REGION Network 1: Режим глобальной симуляции
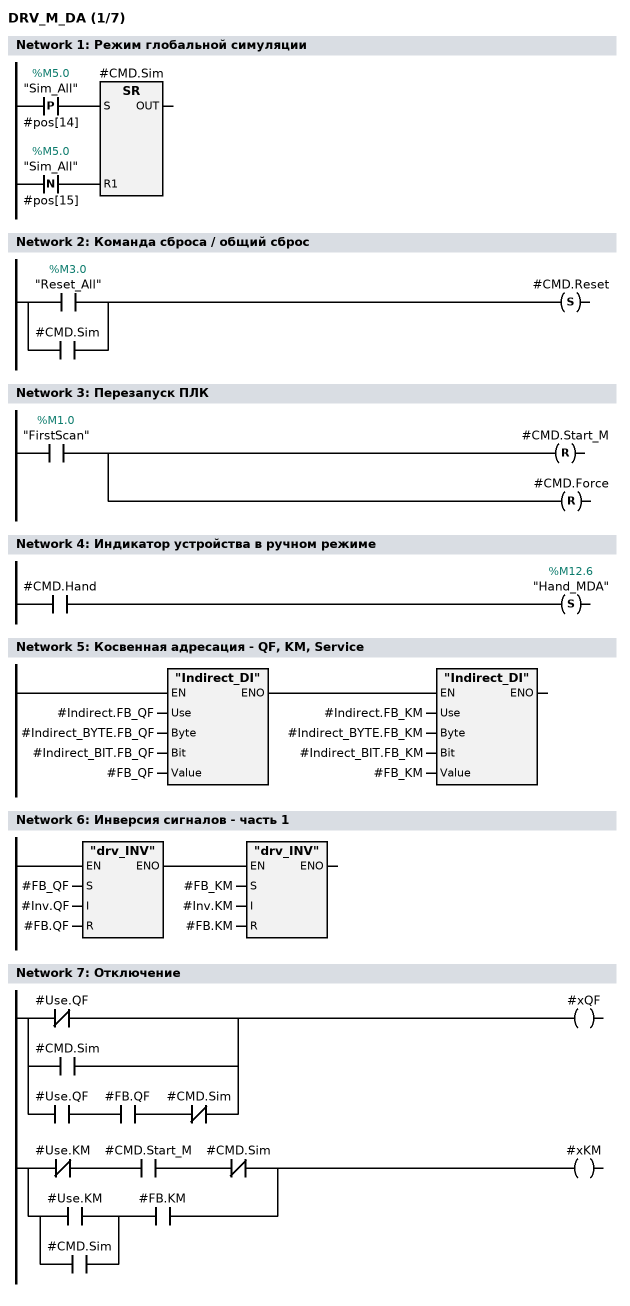
   RUNG wire#powerrail
      P_Contact(operand := "Sim_All", bit := #pos[14])
      S_SR(operand := #CMD.Sim, r1 := wire#w1)
   END_RUNG
   RUNG wire#powerrail
      N_Contact(operand := "Sim_All", bit := #pos[15])
   END_RUNG wire#w1
   // the same network as SCL:
   #_w1 := "Sim_All" AND NOT #pos[14];   // rising edge of "Sim_All"
   #pos[14] := "Sim_All";
   #_w2 := NOT "Sim_All" AND #pos[15];   // falling edge of "Sim_All"
   #pos[15] := "Sim_All";
   IF #_w1 THEN
       #CMD.Sim := TRUE;   // SR flip-flop
   END_IF;
   IF #_w2 THEN #CMD.Sim := FALSE; END_IF;
END_REGION

REGION Network 2: Команда сброса / общий сброс
   RUNG wire#powerrail
      Contact( "Reset_All" )
      wire#w1
      S_Coil( #CMD.Reset )
   END_RUNG
   RUNG wire#powerrail
      Contact( #CMD.Sim )
   END_RUNG wire#w1
   // the same network as SCL:
   IF "Reset_All" OR #CMD.Sim THEN #CMD.Reset := TRUE; END_IF;
END_REGION

REGION Network 3: Перезапуск ПЛК
   RUNG wire#powerrail
      Contact( "FirstScan" )
      wire#w1
      R_Coil( #CMD.Start_M )
   END_RUNG
   RUNG wire#w1
      R_Coil( #CMD.Force )
   END_RUNG
   // the same network as SCL:
   IF "FirstScan" THEN
       #CMD.Start_M := FALSE;
       #CMD.Force := FALSE;
   END_IF;
END_REGION

REGION Network 4: Индикатор устройства в ручном режиме
   RUNG wire#powerrail
      Contact( #CMD.Hand )
      S_Coil( "Hand_MDA" )
   END_RUNG
   // the same network as SCL:
   IF #CMD.Hand THEN "Hand_MDA" := TRUE; END_IF;
END_REGION

REGION Network 5: Косвенная адресация - QF, KM, Service
   RUNG wire#powerrail
      "Indirect_DI"(Use := #Indirect.FB_QF, "Byte" := #Indirect_BYTE.FB_QF, Bit := #Indirect_BIT.FB_QF, Value := #FB_QF)
      "Indirect_DI"(Use := #Indirect.FB_KM, "Byte" := #Indirect_BYTE.FB_KM, Bit := #Indirect_BIT.FB_KM, Value := #FB_KM)
   END_RUNG
   // the same network as SCL:
   "Indirect_DI"(Use := #Indirect.FB_QF,
                 "Byte" := #Indirect_BYTE.FB_QF,
                 Bit := #Indirect_BIT.FB_QF,
                 Value := #FB_QF,
                 ENO => #_w1);
   IF #_w1 THEN
       "Indirect_DI"(Use := #Indirect.FB_KM,
                     "Byte" := #Indirect_BYTE.FB_KM,
                     Bit := #Indirect_BIT.FB_KM,
                     Value := #FB_KM);
   END_IF;
END_REGION

REGION Network 6: Инверсия сигналов - часть 1
   RUNG wire#powerrail
      "drv_INV"(S := #FB_QF, I := #Inv.QF, R := #FB.QF)
      "drv_INV"(S := #FB_KM, I := #Inv.KM, R := #FB.KM)
   END_RUNG
   // the same network as SCL:
   "drv_INV"(S := #FB_QF, I := #Inv.QF, R := #FB.QF, ENO => #_w1);
   IF #_w1 THEN "drv_INV"(S := #FB_KM, I := #Inv.KM, R := #FB.KM); END_IF;
END_REGION

REGION Network 7: Отключение
   RUNG wire#powerrail
      I_Contact( #Use.QF )
      wire#w1
      Coil( #xQF )
   END_RUNG
   RUNG wire#powerrail
      Contact( #CMD.Sim )
   END_RUNG wire#w1
   RUNG wire#powerrail
      Contact( #Use.QF )
      Contact( #FB.QF )
      I_Contact( #CMD.Sim )
   END_RUNG wire#w1
   RUNG wire#powerrail
      I_Contact( #Use.KM )
      Contact( #CMD.Start_M )
      I_Contact( #CMD.Sim )
      wire#w2
      Coil( #xKM )
   END_RUNG
   RUNG wire#powerrail
      Contact( #Use.KM )
      wire#w3
      Contact( #FB.KM )
   END_RUNG wire#w2
   RUNG wire#powerrail
      Contact( #CMD.Sim )
   END_RUNG wire#w3
   // the same network as SCL:
   #xQF := NOT #Use.QF OR #CMD.Sim OR (#Use.QF AND #FB.QF AND NOT #CMD.Sim);
   #xKM := (NOT #Use.KM AND #CMD.Start_M AND NOT #CMD.Sim) OR ((#Use.KM OR #CMD.Sim) AND #FB.KM);
END_REGION

REGION Network 8: Режим работы устройства / определение режима работы
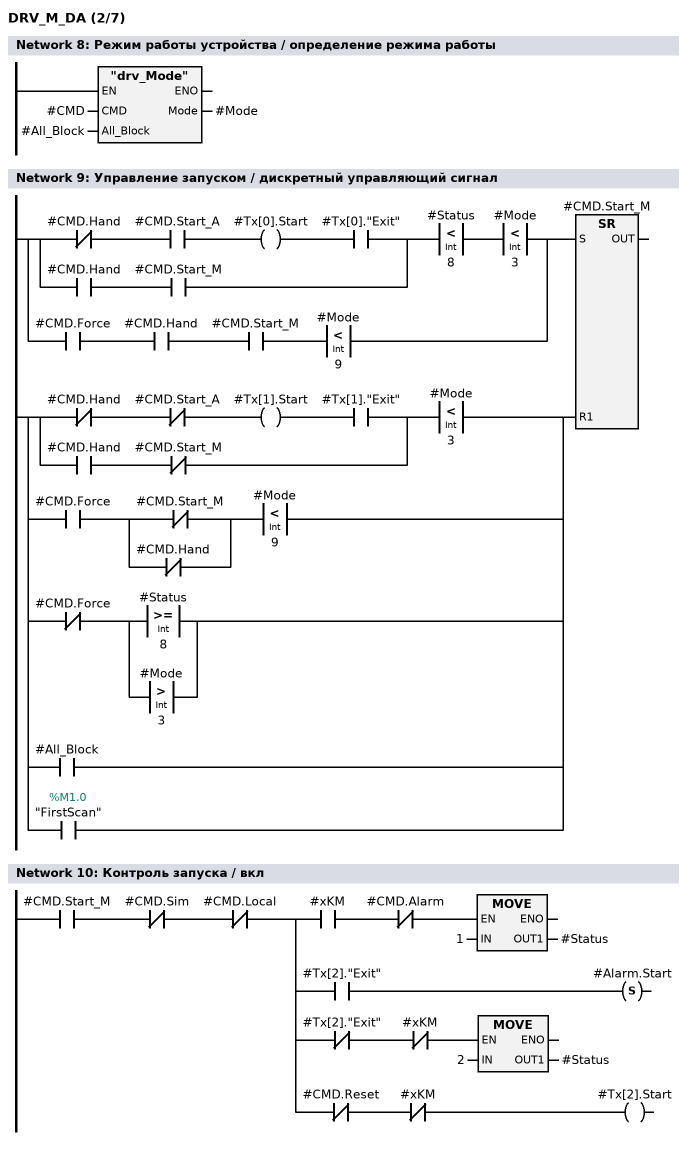
   RUNG wire#powerrail
      "drv_Mode"(CMD := #CMD, All_Block := #All_Block, Mode => #Mode)
   END_RUNG
   // the same network as SCL:
   "drv_Mode"(CMD := #CMD, All_Block := #All_Block, Mode => #Mode);
END_REGION

REGION Network 9: Управление запуском / дискретный управляющий сигнал
   RUNG wire#powerrail
      I_Contact( #CMD.Hand )
      Contact( #CMD.Start_A )
      Coil( #Tx[0].Start )
      Contact( #Tx[0]."Exit" )
      wire#w1
      { S7_Templates := "SrcType := Int" } LT_Contact(in1 := #Status, in2 := 8)
      { S7_Templates := "SrcType := Int" } LT_Contact(in1 := #Mode, in2 := 3)
      wire#w2
      S_SR(operand := #CMD.Start_M, r1 := wire#w7)
   END_RUNG
   RUNG wire#powerrail
      Contact( #CMD.Hand )
      Contact( #CMD.Start_M )
   END_RUNG wire#w1
   RUNG wire#powerrail
      Contact( #CMD.Force )
      Contact( #CMD.Hand )
      Contact( #CMD.Start_M )
      { S7_Templates := "SrcType := Int" } LT_Contact(in1 := #Mode, in2 := 9)
   END_RUNG wire#w2
   RUNG wire#powerrail
      I_Contact( #CMD.Hand )
      I_Contact( #CMD.Start_A )
      Coil( #Tx[1].Start )
      Contact( #Tx[1]."Exit" )
      wire#w3
      { S7_Templates := "SrcType := Int" } LT_Contact(in1 := #Mode, in2 := 3)
   END_RUNG wire#w7
   RUNG wire#powerrail
      Contact( #CMD.Hand )
      I_Contact( #CMD.Start_M )
   END_RUNG wire#w3
   RUNG wire#powerrail
      Contact( #CMD.Force )
      wire#w4
      I_Contact( #CMD.Start_M )
      wire#w5
      { S7_Templates := "SrcType := Int" } LT_Contact(in1 := #Mode, in2 := 9)
   END_RUNG wire#w7
   RUNG wire#w4
      I_Contact( #CMD.Hand )
   END_RUNG wire#w5
   RUNG wire#powerrail
      I_Contact( #CMD.Force )
      wire#w6
      { S7_Templates := "SrcType := Int" } GE_Contact(in1 := #Status, in2 := 8)
   END_RUNG wire#w7
   RUNG wire#w6
      { S7_Templates := "SrcType := Int" } GT_Contact(in1 := #Mode, in2 := 3)
   END_RUNG wire#w7
   RUNG wire#powerrail
      Contact( #All_Block )
   END_RUNG wire#w7
   RUNG wire#powerrail
      Contact( "FirstScan" )
   END_RUNG wire#w7
   // the same network as SCL:
   #Tx[0].Start := NOT #CMD.Hand AND #CMD.Start_A;
   #_w1 := (((NOT #CMD.Hand AND #CMD.Start_A AND #Tx[0]."Exit") OR (#CMD.Hand AND #CMD.Start_M)) AND (#Status < 8) AND (#Mode < 3)) OR (#CMD.Force AND #CMD.Hand AND #CMD.Start_M AND (#Mode < 9));
   #Tx[1].Start := NOT #CMD.Hand AND NOT #CMD.Start_A;
   #_w2 := (((NOT #CMD.Hand AND NOT #CMD.Start_A AND #Tx[1]."Exit") OR (#CMD.Hand AND NOT #CMD.Start_M)) AND (#Mode < 3)) OR (#CMD.Force AND (NOT #CMD.Start_M OR NOT #CMD.Hand) AND (#Mode < 9)) OR (NOT #CMD.Force AND ((#Status >= 8) OR (#Mode > 3))) OR #All_Block OR "FirstScan";
   IF #_w1 THEN
       #CMD.Start_M := TRUE;   // SR flip-flop
   END_IF;
   IF #_w2 THEN #CMD.Start_M := FALSE; END_IF;
END_REGION

REGION Network 10: Контроль запуска / вкл
   RUNG wire#powerrail
      Contact( #CMD.Start_M )
      I_Contact( #CMD.Sim )
      I_Contact( #CMD.Local )
      wire#w1
      Contact( #xKM )
      I_Contact( #CMD.Alarm )
      { S7_GenerateENO := "TRUE" } Move(in := 1, out1 => #Status)
   END_RUNG
   RUNG wire#w1
      Contact( #Tx[2]."Exit" )
      S_Coil( #Alarm.Start )
   END_RUNG
   RUNG wire#w1
      I_Contact( #Tx[2]."Exit" )
      I_Contact( #xKM )
      { S7_GenerateENO := "TRUE" } Move(in := 2, out1 => #Status)
   END_RUNG
   RUNG wire#w1
      I_Contact( #CMD.Reset )
      I_Contact( #xKM )
      Coil( #Tx[2].Start )
   END_RUNG
   // the same network as SCL:
   #_w1 := #CMD.Start_M AND NOT #CMD.Sim AND NOT #CMD.Local;
   IF #_w1 AND #xKM AND NOT #CMD.Alarm THEN #Status := 1; END_IF;
   IF #_w1 AND #Tx[2]."Exit" THEN #Alarm.Start := TRUE; END_IF;
   IF #_w1 AND NOT #Tx[2]."Exit" AND NOT #xKM THEN #Status := 2; END_IF;
   #Tx[2].Start := #_w1 AND NOT #CMD.Reset AND NOT #xKM;
END_REGION

REGION Network 11: Контроль останова / выкл
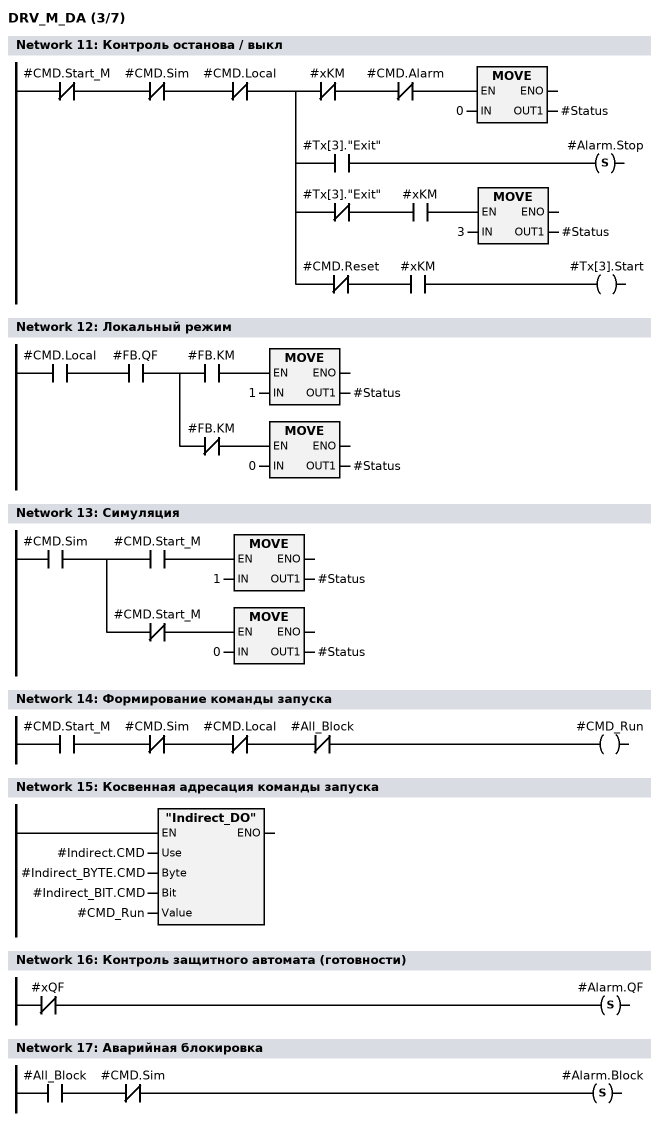
   RUNG wire#powerrail
      I_Contact( #CMD.Start_M )
      I_Contact( #CMD.Sim )
      I_Contact( #CMD.Local )
      wire#w1
      I_Contact( #xKM )
      I_Contact( #CMD.Alarm )
      { S7_GenerateENO := "TRUE" } Move(in := 0, out1 => #Status)
   END_RUNG
   RUNG wire#w1
      Contact( #Tx[3]."Exit" )
      S_Coil( #Alarm.Stop )
   END_RUNG
   RUNG wire#w1
      I_Contact( #Tx[3]."Exit" )
      Contact( #xKM )
      { S7_GenerateENO := "TRUE" } Move(in := 3, out1 => #Status)
   END_RUNG
   RUNG wire#w1
      I_Contact( #CMD.Reset )
      Contact( #xKM )
      Coil( #Tx[3].Start )
   END_RUNG
   // the same network as SCL:
   #_w1 := NOT #CMD.Start_M AND NOT #CMD.Sim AND NOT #CMD.Local;
   IF #_w1 AND NOT #xKM AND NOT #CMD.Alarm THEN #Status := 0; END_IF;
   IF #_w1 AND #Tx[3]."Exit" THEN #Alarm.Stop := TRUE; END_IF;
   IF #_w1 AND NOT #Tx[3]."Exit" AND #xKM THEN #Status := 3; END_IF;
   #Tx[3].Start := #_w1 AND NOT #CMD.Reset AND #xKM;
END_REGION

REGION Network 12: Локальный режим
   RUNG wire#powerrail
      Contact( #CMD.Local )
      Contact( #FB.QF )
      wire#w1
      Contact( #FB.KM )
      { S7_GenerateENO := "TRUE" } Move(in := 1, out1 => #Status)
   END_RUNG
   RUNG wire#w1
      I_Contact( #FB.KM )
      { S7_GenerateENO := "TRUE" } Move(in := 0, out1 => #Status)
   END_RUNG
   // the same network as SCL:
   #_w1 := #CMD.Local AND #FB.QF;
   IF #_w1 AND #FB.KM THEN #Status := 1; END_IF;
   IF #_w1 AND NOT #FB.KM THEN #Status := 0; END_IF;
END_REGION

REGION Network 13: Симуляция
   RUNG wire#powerrail
      Contact( #CMD.Sim )
      wire#w1
      Contact( #CMD.Start_M )
      { S7_GenerateENO := "TRUE" } Move(in := 1, out1 => #Status)
   END_RUNG
   RUNG wire#w1
      I_Contact( #CMD.Start_M )
      { S7_GenerateENO := "TRUE" } Move(in := 0, out1 => #Status)
   END_RUNG
   // the same network as SCL:
   IF #CMD.Sim AND #CMD.Start_M THEN #Status := 1; END_IF;
   IF #CMD.Sim AND NOT #CMD.Start_M THEN #Status := 0; END_IF;
END_REGION

REGION Network 14: Формирование команды запуска
   RUNG wire#powerrail
      Contact( #CMD.Start_M )
      I_Contact( #CMD.Sim )
      I_Contact( #CMD.Local )
      I_Contact( #All_Block )
      Coil( #CMD_Run )
   END_RUNG
   // the same network as SCL:
   #CMD_Run := #CMD.Start_M AND NOT #CMD.Sim AND NOT #CMD.Local AND NOT #All_Block;
END_REGION

REGION Network 15: Косвенная адресация команды запуска
   RUNG wire#powerrail
      "Indirect_DO"(Use := #Indirect.CMD, "Byte" := #Indirect_BYTE.CMD, Bit := #Indirect_BIT.CMD, Value := #CMD_Run)
   END_RUNG
   // the same network as SCL:
   "Indirect_DO"(Use := #Indirect.CMD,
                 "Byte" := #Indirect_BYTE.CMD,
                 Bit := #Indirect_BIT.CMD,
                 Value := #CMD_Run);
END_REGION

REGION Network 16: Контроль защитного автомата (готовности)
   RUNG wire#powerrail
      I_Contact( #xQF )
      S_Coil( #Alarm.QF )
   END_RUNG
   // the same network as SCL:
   IF NOT #xQF THEN #Alarm.QF := TRUE; END_IF;
END_REGION

REGION Network 17: Аварийная блокировка
   RUNG wire#powerrail
      Contact( #All_Block )
      I_Contact( #CMD.Sim )
      S_Coil( #Alarm.Block )
   END_RUNG
   // the same network as SCL:
   IF #All_Block AND NOT #CMD.Sim THEN #Alarm.Block := TRUE; END_IF;
END_REGION

REGION Network 18: Сигнал аварии
   // Safety - сработал датчик безопасности, подключается через отдельный дискретный вход
   // Termo - сработала термозащита, подключается через отдельный дискретный вход
   // Alarm - сработала внешняя авария, подключается через отдельный дискретный вход
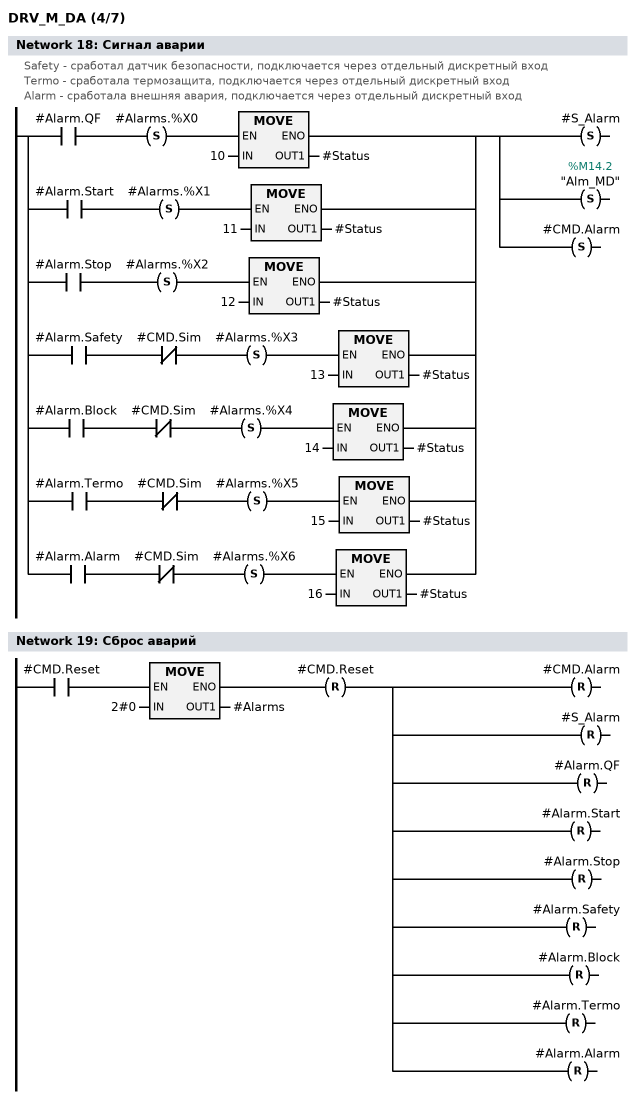
   RUNG wire#powerrail
      Contact( #Alarm.QF )
      S_Coil( #Alarms.%X0 )
      { S7_GenerateENO := "TRUE" } Move(in := 10, out1 => #Status)
      wire#w1
      S_Coil( #S_Alarm )
   END_RUNG
   RUNG wire#powerrail
      Contact( #Alarm.Start )
      S_Coil( #Alarms.%X1 )
      { S7_GenerateENO := "TRUE" } Move(in := 11, out1 => #Status)
   END_RUNG wire#w1
   RUNG wire#powerrail
      Contact( #Alarm.Stop )
      S_Coil( #Alarms.%X2 )
      { S7_GenerateENO := "TRUE" } Move(in := 12, out1 => #Status)
   END_RUNG wire#w1
   RUNG wire#powerrail
      Contact( #Alarm.Safety )
      I_Contact( #CMD.Sim )
      S_Coil( #Alarms.%X3 )
      { S7_GenerateENO := "TRUE" } Move(in := 13, out1 => #Status)
   END_RUNG wire#w1
   RUNG wire#powerrail
      Contact( #Alarm.Block )
      I_Contact( #CMD.Sim )
      S_Coil( #Alarms.%X4 )
      { S7_GenerateENO := "TRUE" } Move(in := 14, out1 => #Status)
   END_RUNG wire#w1
   RUNG wire#powerrail
      Contact( #Alarm.Termo )
      I_Contact( #CMD.Sim )
      S_Coil( #Alarms.%X5 )
      { S7_GenerateENO := "TRUE" } Move(in := 15, out1 => #Status)
   END_RUNG wire#w1
   RUNG wire#powerrail
      Contact( #Alarm.Alarm )
      I_Contact( #CMD.Sim )
      S_Coil( #Alarms.%X6 )
      { S7_GenerateENO := "TRUE" } Move(in := 16, out1 => #Status)
   END_RUNG wire#w1
   RUNG wire#w1
      S_Coil( "Alm_MD" )
   END_RUNG
   RUNG wire#w1
      S_Coil( #CMD.Alarm )
   END_RUNG
   // the same network as SCL:
   // ENO of a box is taken as its EN; it also drops when the box reports an error
   IF #Alarm.QF THEN
       #Alarms.%X0 := TRUE;
       #Status := 10;
   END_IF;
   IF #Alarm.Start THEN
       #Alarms.%X1 := TRUE;
       #Status := 11;
   END_IF;
   IF #Alarm.Stop THEN
       #Alarms.%X2 := TRUE;
       #Status := 12;
   END_IF;
   #_w1 := #Alarm.Safety AND NOT #CMD.Sim;
   IF #_w1 THEN
       #Alarms.%X3 := TRUE;
       #Status := 13;
   END_IF;
   #_w2 := #Alarm.Block AND NOT #CMD.Sim;
   IF #_w2 THEN
       #Alarms.%X4 := TRUE;
       #Status := 14;
   END_IF;
   #_w3 := #Alarm.Termo AND NOT #CMD.Sim;
   IF #_w3 THEN
       #Alarms.%X5 := TRUE;
       #Status := 15;
   END_IF;
   #_w4 := #Alarm.Alarm AND NOT #CMD.Sim;
   IF #_w4 THEN
       #Alarms.%X6 := TRUE;
       #Status := 16;
   END_IF;
   IF #Alarm.QF OR #Alarm.Start OR #Alarm.Stop OR #_w1 OR #_w2 OR #_w3 OR #_w4 THEN
       #S_Alarm := TRUE;
       "Alm_MD" := TRUE;
       #CMD.Alarm := TRUE;
   END_IF;
END_REGION

REGION Network 19: Сброс аварий
   RUNG wire#powerrail
      Contact( #CMD.Reset )
      Move(in := 2#0, out1 => #Alarms)
      R_Coil( #CMD.Reset )
      wire#w1
      R_Coil( #CMD.Alarm )
   END_RUNG
   RUNG wire#w1
      R_Coil( #S_Alarm )
   END_RUNG
   RUNG wire#w1
      R_Coil( #Alarm.QF )
   END_RUNG
   RUNG wire#w1
      R_Coil( #Alarm.Start )
   END_RUNG
   RUNG wire#w1
      R_Coil( #Alarm.Stop )
   END_RUNG
   RUNG wire#w1
      R_Coil( #Alarm.Safety )
   END_RUNG
   RUNG wire#w1
      R_Coil( #Alarm.Block )
   END_RUNG
   RUNG wire#w1
      R_Coil( #Alarm.Termo )
   END_RUNG
   RUNG wire#w1
      R_Coil( #Alarm.Alarm )
   END_RUNG
   // the same network as SCL:
   IF #CMD.Reset THEN #Alarms := 2#0; END_IF;
   #_w1 := #CMD.Reset;
   IF #_w1 THEN
       #CMD.Reset := FALSE;
       #CMD.Alarm := FALSE;
       #S_Alarm := FALSE;
       #Alarm.QF := FALSE;
       #Alarm.Start := FALSE;
       #Alarm.Stop := FALSE;
       #Alarm.Safety := FALSE;
       #Alarm.Block := FALSE;
       #Alarm.Termo := FALSE;
       #Alarm.Alarm := FALSE;
   END_IF;
END_REGION

REGION Network 20: События привода
   // 0 - ручной режим активирован
   // 1 - ручной режим деактивирован
   // 2 - принудительный режим активирован
   // 3 - принудительный режим деактивирован
   // 4 - запуск в ручном режиме
   // 5 - останов в ручном режиме
   // 6 - местный режим управления активирован
   // 7 - местный режим управления деактивирован
   // 8 - запущено в местном режиме
   // 9 - остановлено в местном режиме
   // 10 - сервисный режим активирован
   // 11 - сервисный режим деактивирован
   // 12 - проведено сервисное обслуживание
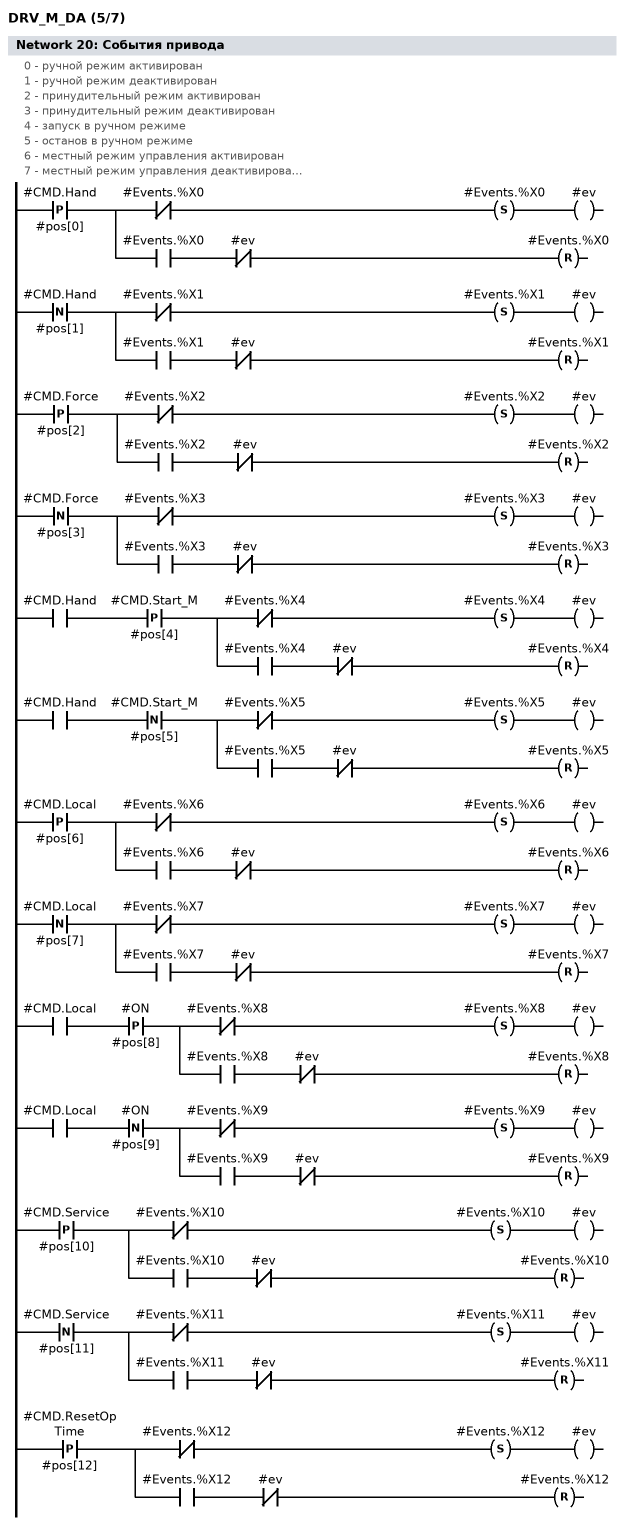
   RUNG wire#powerrail
      P_Contact(operand := #CMD.Hand, bit := #pos[0])
      wire#w1
      I_Contact( #Events.%X0 )
      S_Coil( #Events.%X0 )
      Coil( #ev )
   END_RUNG
   RUNG wire#w1
      Contact( #Events.%X0 )
      I_Contact( #ev )
      R_Coil( #Events.%X0 )
   END_RUNG
   RUNG wire#powerrail
      N_Contact(operand := #CMD.Hand, bit := #pos[1])
      wire#w2
      I_Contact( #Events.%X1 )
      S_Coil( #Events.%X1 )
      Coil( #ev )
   END_RUNG
   RUNG wire#w2
      Contact( #Events.%X1 )
      I_Contact( #ev )
      R_Coil( #Events.%X1 )
   END_RUNG
   RUNG wire#powerrail
      P_Contact(operand := #CMD.Force, bit := #pos[2])
      wire#w3
      I_Contact( #Events.%X2 )
      S_Coil( #Events.%X2 )
      Coil( #ev )
   END_RUNG
   RUNG wire#w3
      Contact( #Events.%X2 )
      I_Contact( #ev )
      R_Coil( #Events.%X2 )
   END_RUNG
   RUNG wire#powerrail
      N_Contact(operand := #CMD.Force, bit := #pos[3])
      wire#w4
      I_Contact( #Events.%X3 )
      S_Coil( #Events.%X3 )
      Coil( #ev )
   END_RUNG
   RUNG wire#w4
      Contact( #Events.%X3 )
      I_Contact( #ev )
      R_Coil( #Events.%X3 )
   END_RUNG
   RUNG wire#powerrail
      Contact( #CMD.Hand )
      P_Contact(operand := #CMD.Start_M, bit := #pos[4])
      wire#w5
      I_Contact( #Events.%X4 )
      S_Coil( #Events.%X4 )
      Coil( #ev )
   END_RUNG
   RUNG wire#w5
      Contact( #Events.%X4 )
      I_Contact( #ev )
      R_Coil( #Events.%X4 )
   END_RUNG
   RUNG wire#powerrail
      Contact( #CMD.Hand )
      N_Contact(operand := #CMD.Start_M, bit := #pos[5])
      wire#w6
      I_Contact( #Events.%X5 )
      S_Coil( #Events.%X5 )
      Coil( #ev )
   END_RUNG
   RUNG wire#w6
      Contact( #Events.%X5 )
      I_Contact( #ev )
      R_Coil( #Events.%X5 )
   END_RUNG
   RUNG wire#powerrail
      P_Contact(operand := #CMD.Local, bit := #pos[6])
      wire#w7
      I_Contact( #Events.%X6 )
      S_Coil( #Events.%X6 )
      Coil( #ev )
   END_RUNG
   RUNG wire#w7
      Contact( #Events.%X6 )
      I_Contact( #ev )
      R_Coil( #Events.%X6 )
   END_RUNG
   RUNG wire#powerrail
      N_Contact(operand := #CMD.Local, bit := #pos[7])
      wire#w8
      I_Contact( #Events.%X7 )
      S_Coil( #Events.%X7 )
      Coil( #ev )
   END_RUNG
   RUNG wire#w8
      Contact( #Events.%X7 )
      I_Contact( #ev )
      R_Coil( #Events.%X7 )
   END_RUNG
   RUNG wire#powerrail
      Contact( #CMD.Local )
      P_Contact(operand := #ON, bit := #pos[8])
      wire#w9
      I_Contact( #Events.%X8 )
      S_Coil( #Events.%X8 )
      Coil( #ev )
   END_RUNG
   RUNG wire#w9
      Contact( #Events.%X8 )
      I_Contact( #ev )
      R_Coil( #Events.%X8 )
   END_RUNG
   RUNG wire#powerrail
      Contact( #CMD.Local )
      N_Contact(operand := #ON, bit := #pos[9])
      wire#w10
      I_Contact( #Events.%X9 )
      S_Coil( #Events.%X9 )
      Coil( #ev )
   END_RUNG
   RUNG wire#w10
      Contact( #Events.%X9 )
      I_Contact( #ev )
      R_Coil( #Events.%X9 )
   END_RUNG
   RUNG wire#powerrail
      P_Contact(operand := #CMD.Service, bit := #pos[10])
      wire#w11
      I_Contact( #Events.%X10 )
      S_Coil( #Events.%X10 )
      Coil( #ev )
   END_RUNG
   RUNG wire#w11
      Contact( #Events.%X10 )
      I_Contact( #ev )
      R_Coil( #Events.%X10 )
   END_RUNG
   RUNG wire#powerrail
      N_Contact(operand := #CMD.Service, bit := #pos[11])
      wire#w12
      I_Contact( #Events.%X11 )
      S_Coil( #Events.%X11 )
      Coil( #ev )
   END_RUNG
   RUNG wire#w12
      Contact( #Events.%X11 )
      I_Contact( #ev )
      R_Coil( #Events.%X11 )
   END_RUNG
   RUNG wire#powerrail
      P_Contact(operand := #CMD.ResetOpTime, bit := #pos[12])
      wire#w13
      I_Contact( #Events.%X12 )
      S_Coil( #Events.%X12 )
      Coil( #ev )
   END_RUNG
   RUNG wire#w13
      Contact( #Events.%X12 )
      I_Contact( #ev )
      R_Coil( #Events.%X12 )
   END_RUNG
   // the same network as SCL:
   #_w1 := #CMD.Hand AND NOT #pos[0];   // rising edge of #CMD.Hand
   #pos[0] := #CMD.Hand;
   #_w2 := #_w1 AND NOT #Events.%X0;
   IF #_w2 THEN #Events.%X0 := TRUE; END_IF;
   #ev := #_w2;
   IF #_w1 AND #Events.%X0 AND NOT #ev THEN #Events.%X0 := FALSE; END_IF;
   #_w3 := NOT #CMD.Hand AND #pos[1];   // falling edge of #CMD.Hand
   #pos[1] := #CMD.Hand;
   #_w4 := #_w3 AND NOT #Events.%X1;
   IF #_w4 THEN #Events.%X1 := TRUE; END_IF;
   #ev := #_w4;
   IF #_w3 AND #Events.%X1 AND NOT #ev THEN #Events.%X1 := FALSE; END_IF;
   #_w5 := #CMD.Force AND NOT #pos[2];   // rising edge of #CMD.Force
   #pos[2] := #CMD.Force;
   #_w6 := #_w5 AND NOT #Events.%X2;
   IF #_w6 THEN #Events.%X2 := TRUE; END_IF;
   #ev := #_w6;
   IF #_w5 AND #Events.%X2 AND NOT #ev THEN #Events.%X2 := FALSE; END_IF;
   #_w7 := NOT #CMD.Force AND #pos[3];   // falling edge of #CMD.Force
   #pos[3] := #CMD.Force;
   #_w8 := #_w7 AND NOT #Events.%X3;
   IF #_w8 THEN #Events.%X3 := TRUE; END_IF;
   #ev := #_w8;
   IF #_w7 AND #Events.%X3 AND NOT #ev THEN #Events.%X3 := FALSE; END_IF;
   #_w9 := #CMD.Hand AND #CMD.Start_M AND NOT #pos[4];   // rising edge of #CMD.Start_M
   #pos[4] := #CMD.Start_M;
   #_w10 := #_w9 AND NOT #Events.%X4;
   IF #_w10 THEN #Events.%X4 := TRUE; END_IF;
   #ev := #_w10;
   IF #_w9 AND #Events.%X4 AND NOT #ev THEN #Events.%X4 := FALSE; END_IF;
   #_w11 := #CMD.Hand AND NOT #CMD.Start_M AND #pos[5];   // falling edge of #CMD.Start_M
   #pos[5] := #CMD.Start_M;
   #_w12 := #_w11 AND NOT #Events.%X5;
   IF #_w12 THEN #Events.%X5 := TRUE; END_IF;
   #ev := #_w12;
   IF #_w11 AND #Events.%X5 AND NOT #ev THEN #Events.%X5 := FALSE; END_IF;
   #_w13 := #CMD.Local AND NOT #pos[6];   // rising edge of #CMD.Local
   #pos[6] := #CMD.Local;
   #_w14 := #_w13 AND NOT #Events.%X6;
   IF #_w14 THEN #Events.%X6 := TRUE; END_IF;
   #ev := #_w14;
   IF #_w13 AND #Events.%X6 AND NOT #ev THEN #Events.%X6 := FALSE; END_IF;
   #_w15 := NOT #CMD.Local AND #pos[7];   // falling edge of #CMD.Local
   #pos[7] := #CMD.Local;
   #_w16 := #_w15 AND NOT #Events.%X7;
   IF #_w16 THEN #Events.%X7 := TRUE; END_IF;
   #ev := #_w16;
   IF #_w15 AND #Events.%X7 AND NOT #ev THEN #Events.%X7 := FALSE; END_IF;
   #_w17 := #CMD.Local AND #ON AND NOT #pos[8];   // rising edge of #ON
   #pos[8] := #ON;
   #_w18 := #_w17 AND NOT #Events.%X8;
   IF #_w18 THEN #Events.%X8 := TRUE; END_IF;
   #ev := #_w18;
   IF #_w17 AND #Events.%X8 AND NOT #ev THEN #Events.%X8 := FALSE; END_IF;
   #_w19 := #CMD.Local AND NOT #ON AND #pos[9];   // falling edge of #ON
   #pos[9] := #ON;
   #_w20 := #_w19 AND NOT #Events.%X9;
   IF #_w20 THEN #Events.%X9 := TRUE; END_IF;
   #ev := #_w20;
   IF #_w19 AND #Events.%X9 AND NOT #ev THEN #Events.%X9 := FALSE; END_IF;
   #_w21 := #CMD.Service AND NOT #pos[10];   // rising edge of #CMD.Service
   #pos[10] := #CMD.Service;
   #_w22 := #_w21 AND NOT #Events.%X10;
   IF #_w22 THEN #Events.%X10 := TRUE; END_IF;
   #ev := #_w22;
   IF #_w21 AND #Events.%X10 AND NOT #ev THEN #Events.%X10 := FALSE; END_IF;
   #_w23 := NOT #CMD.Service AND #pos[11];   // falling edge of #CMD.Service
   #pos[11] := #CMD.Service;
   #_w24 := #_w23 AND NOT #Events.%X11;
   IF #_w24 THEN #Events.%X11 := TRUE; END_IF;
   #ev := #_w24;
   IF #_w23 AND #Events.%X11 AND NOT #ev THEN #Events.%X11 := FALSE; END_IF;
   #_w25 := #CMD.ResetOpTime AND NOT #pos[12];   // rising edge of #CMD.ResetOpTime
   #pos[12] := #CMD.ResetOpTime;
   #_w26 := #_w25 AND NOT #Events.%X12;
   IF #_w26 THEN #Events.%X12 := TRUE; END_IF;
   #ev := #_w26;
   IF #_w25 AND #Events.%X12 AND NOT #ev THEN #Events.%X12 := FALSE; END_IF;
END_REGION

REGION Network 21: Сервисный режим
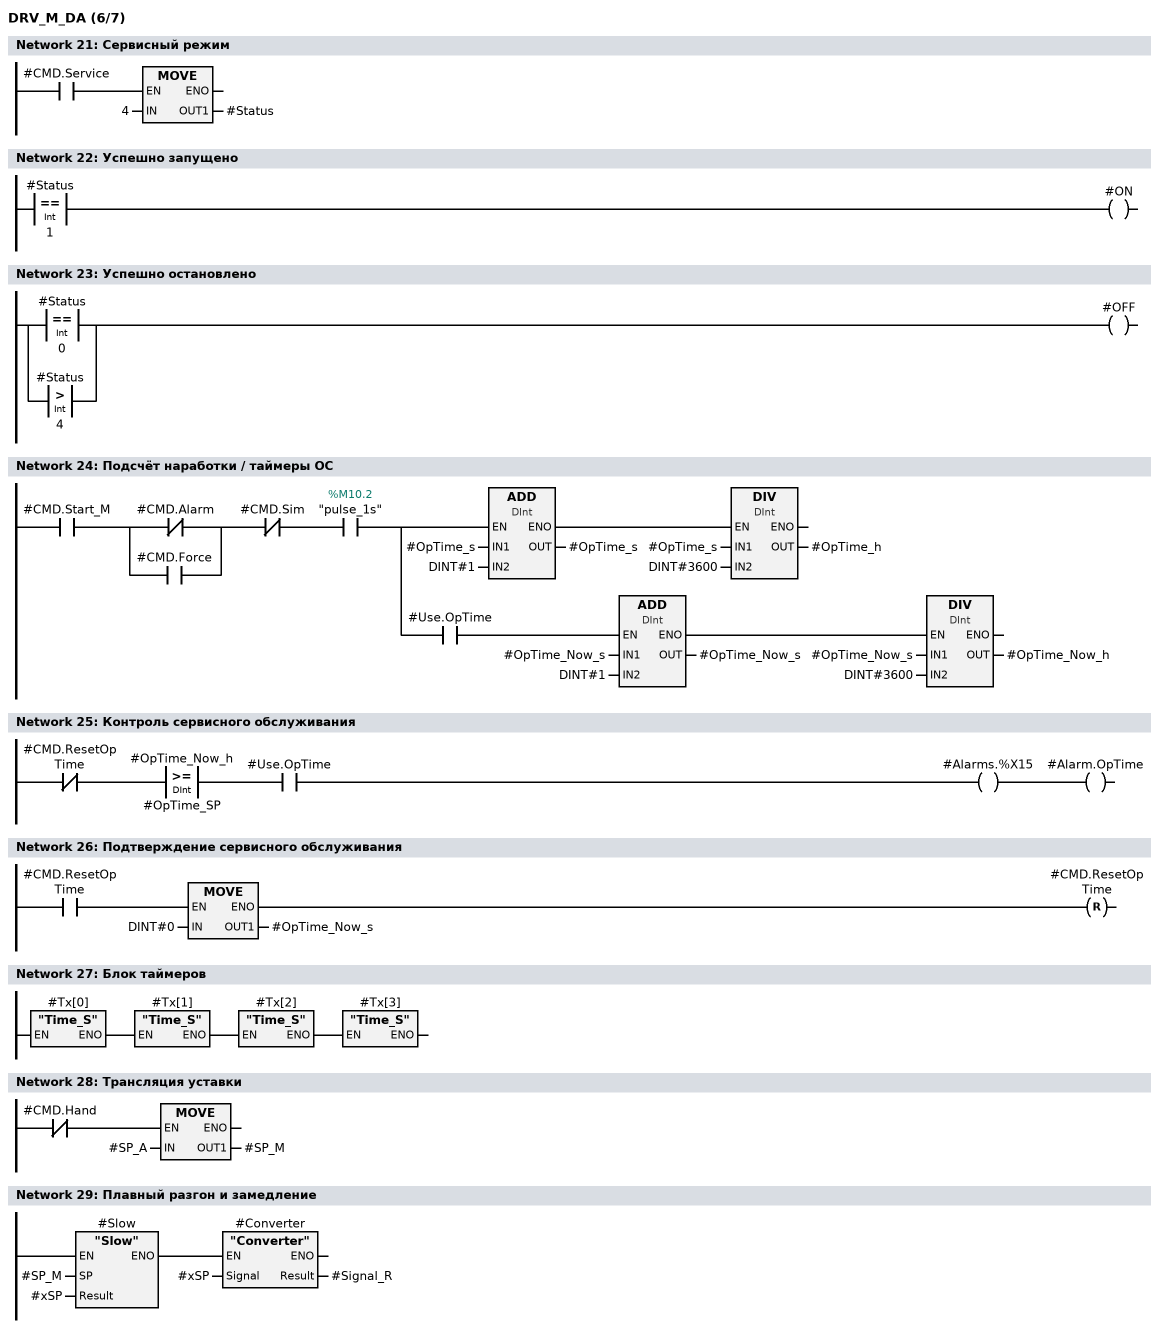
   RUNG wire#powerrail
      Contact( #CMD.Service )
      { S7_GenerateENO := "TRUE" } Move(in := 4, out1 => #Status)
   END_RUNG
   // the same network as SCL:
   IF #CMD.Service THEN #Status := 4; END_IF;
END_REGION

REGION Network 22: Успешно запущено
   RUNG wire#powerrail
      { S7_Templates := "SrcType := Int" } EQ_Contact(in1 := #Status, in2 := 1)
      Coil( #ON )
   END_RUNG
   // the same network as SCL:
   #ON := #Status = 1;
END_REGION

REGION Network 23: Успешно остановлено
   RUNG wire#powerrail
      { S7_Templates := "SrcType := Int" } EQ_Contact(in1 := #Status, in2 := 0)
      wire#w1
      Coil( #OFF )
   END_RUNG
   RUNG wire#powerrail
      { S7_Templates := "SrcType := Int" } GT_Contact(in1 := #Status, in2 := 4)
   END_RUNG wire#w1
   // the same network as SCL:
   #OFF := (#Status = 0) OR (#Status > 4);
END_REGION

REGION Network 24: Подсчёт наработки / таймеры ОС
   RUNG wire#powerrail
      Contact( #CMD.Start_M )
      wire#w1
      I_Contact( #CMD.Alarm )
      wire#w2
      I_Contact( #CMD.Sim )
      Contact( "pulse_1s" )
      wire#w3
      { S7_Templates := "SrcType := DInt"; S7_GenerateENO := "TRUE" } Add(in1 := #OpTime_s, in2 := DINT#1, out => #OpTime_s)
      { S7_Templates := "SrcType := DInt"; S7_GenerateENO := "TRUE" } Div(in1 := #OpTime_s, in2 := DINT#3600, out => #OpTime_h)
   END_RUNG
   RUNG wire#w1
      Contact( #CMD.Force )
   END_RUNG wire#w2
   RUNG wire#w3
      Contact( #Use.OpTime )
      { S7_Templates := "SrcType := DInt"; S7_GenerateENO := "TRUE" } Add(in1 := #OpTime_Now_s, in2 := DINT#1, out => #OpTime_Now_s)
      { S7_Templates := "SrcType := DInt"; S7_GenerateENO := "TRUE" } Div(in1 := #OpTime_Now_s, in2 := DINT#3600, out => #OpTime_Now_h)
   END_RUNG
   // the same network as SCL:
   // ENO of a box is taken as its EN; it also drops when the box reports an error
   #_w1 := #CMD.Start_M AND (NOT #CMD.Alarm OR #CMD.Force) AND NOT #CMD.Sim AND "pulse_1s";
   IF #_w1 THEN
       #OpTime_s := #OpTime_s + DINT#1;
       #OpTime_h := #OpTime_s / DINT#3600;
   END_IF;
   IF #_w1 AND #Use.OpTime THEN
       #OpTime_Now_s := #OpTime_Now_s + DINT#1;
       #OpTime_Now_h := #OpTime_Now_s / DINT#3600;
   END_IF;
END_REGION

REGION Network 25: Контроль сервисного обслуживания
   RUNG wire#powerrail
      I_Contact( #CMD.ResetOpTime )
      { S7_Templates := "SrcType := DInt" } GE_Contact(in1 := #OpTime_Now_h, in2 := #OpTime_SP)
      Contact( #Use.OpTime )
      Coil( #Alarms.%X15 )
      Coil( #Alarm.OpTime )
   END_RUNG
   // the same network as SCL:
   #Alarms.%X15 := NOT #CMD.ResetOpTime AND (#OpTime_Now_h >= #OpTime_SP) AND #Use.OpTime;
   #Alarm.OpTime := #Alarms.%X15;
END_REGION

REGION Network 26: Подтверждение сервисного обслуживания
   RUNG wire#powerrail
      Contact( #CMD.ResetOpTime )
      { S7_GenerateENO := "TRUE" } Move(in := DINT#0, out1 => #OpTime_Now_s)
      R_Coil( #CMD.ResetOpTime )
   END_RUNG
   // the same network as SCL:
   // ENO of a box is taken as its EN; it also drops when the box reports an error
   IF #CMD.ResetOpTime THEN
       #OpTime_Now_s := DINT#0;
       #CMD.ResetOpTime := FALSE;
   END_IF;
END_REGION

REGION Network 27: Блок таймеров
   RUNG wire#powerrail
      #Tx[0]()
      #Tx[1]()
      #Tx[2]()
      #Tx[3]()
   END_RUNG
   // the same network as SCL:
   #Tx[0](ENO => #_w1);   // "Time_S"
   #Tx[1](EN := #_w1, ENO => #_w2);   // "Time_S"
   #Tx[2](EN := #_w2, ENO => #_w3);   // "Time_S"
   IF #_w3 THEN
       #Tx[3]();   // "Time_S"
   END_IF;
END_REGION

REGION Network 28: Трансляция уставки
   RUNG wire#powerrail
      I_Contact( #CMD.Hand )
      Move(in := #SP_A, out1 => #SP_M)
   END_RUNG
   // the same network as SCL:
   IF NOT #CMD.Hand THEN #SP_M := #SP_A; END_IF;
END_REGION

REGION Network 29: Плавный разгон и замедление
   RUNG wire#powerrail
      #Slow(SP := #SP_M, Result := #xSP)
      #Converter(Signal := #xSP, Result => #Signal_R)
   END_RUNG
   // the same network as SCL:
   #Slow(SP := #SP_M, Result := #xSP, ENO => #_w1);   // "Slow"
   IF #_w1 THEN
       #Converter(Signal := #xSP, Result => #Signal_R);   // "Converter"
   END_IF;
END_REGION

REGION Network 30: Выходной аналоговый сигнал
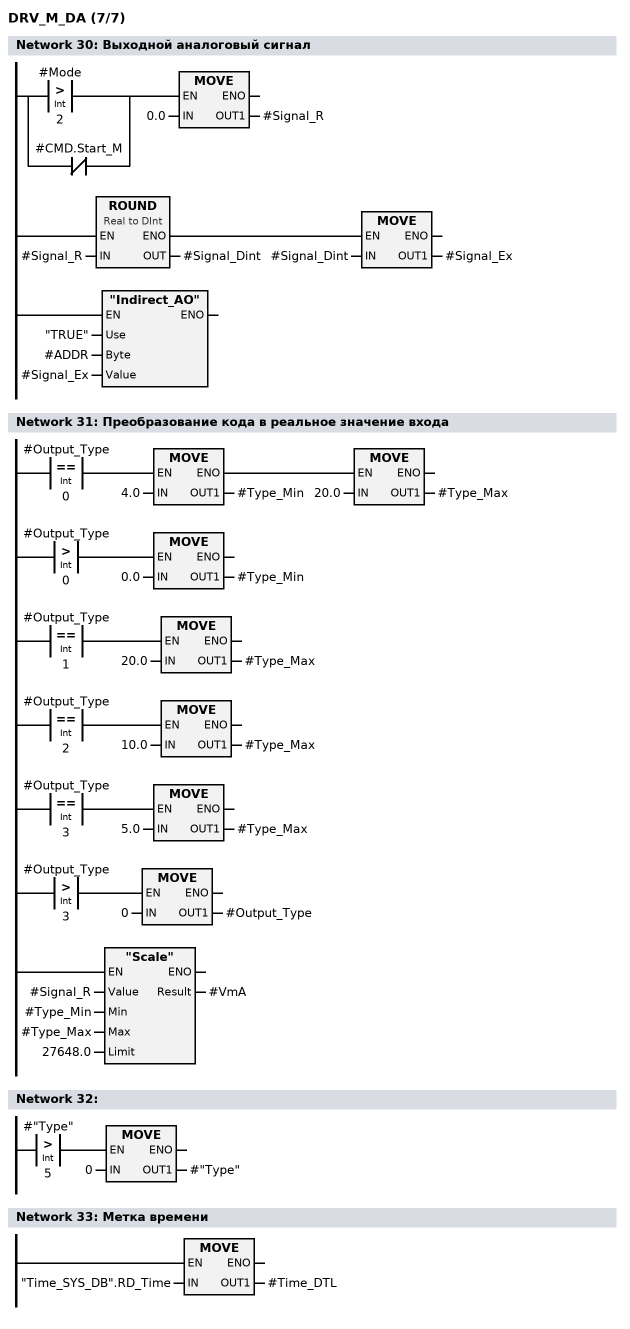
   RUNG wire#powerrail
      { S7_Templates := "SrcType := Int" } GT_Contact(in1 := #Mode, in2 := 2)
      wire#w1
      Move(in := 0.0, out1 => #Signal_R)
   END_RUNG
   RUNG wire#powerrail
      I_Contact( #CMD.Start_M )
   END_RUNG wire#w1
   RUNG wire#powerrail
      { S7_Templates := "[SrcType := Real, DestType := DInt]"; S7_GenerateENO := "TRUE" } Round(in := #Signal_R, out => #Signal_Dint)
      Move(in := #Signal_Dint, out1 => #Signal_Ex)
   END_RUNG
   RUNG wire#powerrail
      "Indirect_AO"(Use := "TRUE", "Byte" := #ADDR, Value := #Signal_Ex)
   END_RUNG
   // the same network as SCL:
   // ENO of a box is taken as its EN; it also drops when the box reports an error
   IF (#Mode > 2) OR NOT #CMD.Start_M THEN #Signal_R := 0.0; END_IF;
   #Signal_Dint := ROUND(#Signal_R);
   #Signal_Ex := #Signal_Dint;
   "Indirect_AO"(Use := "TRUE", "Byte" := #ADDR, Value := #Signal_Ex);
END_REGION

REGION Network 31: Преобразование кода в реальное значение входа
   RUNG wire#powerrail
      { S7_Templates := "SrcType := Int" } EQ_Contact(in1 := #Output_Type, in2 := 0)
      Move(in := 4.0, out1 => #Type_Min)
      Move(in := 20.0, out1 => #Type_Max)
   END_RUNG
   RUNG wire#powerrail
      { S7_Templates := "SrcType := Int" } GT_Contact(in1 := #Output_Type, in2 := 0)
      Move(in := 0.0, out1 => #Type_Min)
   END_RUNG
   RUNG wire#powerrail
      { S7_Templates := "SrcType := Int" } EQ_Contact(in1 := #Output_Type, in2 := 1)
      Move(in := 20.0, out1 => #Type_Max)
   END_RUNG
   RUNG wire#powerrail
      { S7_Templates := "SrcType := Int" } EQ_Contact(in1 := #Output_Type, in2 := 2)
      Move(in := 10.0, out1 => #Type_Max)
   END_RUNG
   RUNG wire#powerrail
      { S7_Templates := "SrcType := Int" } EQ_Contact(in1 := #Output_Type, in2 := 3)
      Move(in := 5.0, out1 => #Type_Max)
   END_RUNG
   RUNG wire#powerrail
      { S7_Templates := "SrcType := Int" } GT_Contact(in1 := #Output_Type, in2 := 3)
      Move(in := 0, out1 => #Output_Type)
   END_RUNG
   RUNG wire#powerrail
      "Scale"(Value := #Signal_R, Min := #Type_Min, Max := #Type_Max, Limit := 27648.0, Result => #VmA)
   END_RUNG
   // the same network as SCL:
   IF #Output_Type = 0 THEN
       #Type_Min := 4.0;
       #Type_Max := 20.0;
   END_IF;
   IF #Output_Type > 0 THEN #Type_Min := 0.0; END_IF;
   IF #Output_Type = 1 THEN #Type_Max := 20.0; END_IF;
   IF #Output_Type = 2 THEN #Type_Max := 10.0; END_IF;
   IF #Output_Type = 3 THEN #Type_Max := 5.0; END_IF;
   IF #Output_Type > 3 THEN #Output_Type := 0; END_IF;
   "Scale"(Value := #Signal_R, Min := #Type_Min, Max := #Type_Max, Limit := 27648.0, Result => #VmA);
END_REGION

REGION Network 32
   RUNG wire#powerrail
      { S7_Templates := "SrcType := Int" } GT_Contact(in1 := #"Type", in2 := 5)
      Move(in := 0, out1 => #"Type")
   END_RUNG
   // the same network as SCL:
   IF #"Type" > 5 THEN #"Type" := 0; END_IF;
END_REGION

REGION Network 33: Метка времени
   RUNG wire#powerrail
      Move(in := "Time_SYS_DB".RD_Time, out1 => #Time_DTL)
   END_RUNG
   // the same network as SCL:
   #Time_DTL := "Time_SYS_DB".RD_Time;
END_REGION
END_FUNCTION_BLOCK

FUNCTION_BLOCK "Valves"   // FB250, LAD
TITLE = Клапана
{ S7_Optimized_Access := 'FALSE' }
VERSION : 0.1
// FB_Alarm - аварийный сигнал для отключения клапана (например по давлению воздуха), 0 - авария, 1 - норма
// FB_QF - сигнал готовности к работе (например, по наличию 24в в линии управления пневмораспределителем), 0 - авария, 1 - норма
// FB_Open - обратная связь датчика открытия клапана, 0 - закрыт, 1 - открыт
// FB_Close - обратная связь датчика закрытия клапана, 1 - закрыт, 0 - открыт
// Value - управление аналоговым клапаном с позиционированием, формат Real, передаётся в блок AO_ex для конвертации в выходной сигнал контроллера (PQW), для использования установите #CMD.Analog в True
// 
// Q -  постоянный сигнал управления клапаном, 0 - закрыть, 1 - открыть
// stored: AutoNumber false, IsIECCheckEnabled false, SetENOAutomatically false, UDAEnableTagReadback false
   VAR DB_SPECIFIC
      Time_DTL { S7_SetPoint := 'True'} : DTL;
   END_VAR
   VAR_TEMP   // added for the SCL form of the ladder/FBD networks
      _w1 : Bool;
   END_VAR
BEGIN

REGION Network 1: Задвижки
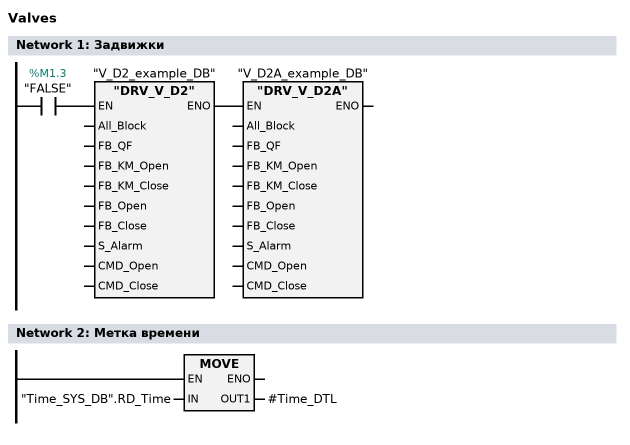
   RUNG wire#powerrail
      Contact( "FALSE" )
      "V_D2_example_DB"(All_Block :=, FB_QF :=, FB_KM_Open :=, FB_KM_Close :=, FB_Open :=, FB_Close :=, S_Alarm :=, CMD_Open :=, CMD_Close :=)
      "V_D2A_example_DB"(All_Block :=, FB_QF :=, FB_KM_Open :=, FB_KM_Close :=, FB_Open :=, FB_Close :=, S_Alarm :=, CMD_Open :=, CMD_Close :=)
   END_RUNG
   // the same network as SCL:
   "V_D2_example_DB"(EN := "FALSE", ENO => #_w1);   // "DRV_V_D2"
   IF #_w1 THEN
       "V_D2A_example_DB"();   // "DRV_V_D2A"
   END_IF;
END_REGION

REGION Network 2: Метка времени
   RUNG wire#powerrail
      Move(in := "Time_SYS_DB".RD_Time, out1 => #Time_DTL)
   END_RUNG
   // the same network as SCL:
   #Time_DTL := "Time_SYS_DB".RD_Time;
END_REGION
END_FUNCTION_BLOCK

FUNCTION_BLOCK "DRV_V_D2"   // FB120, LAD
TITLE = Управление клапаном с двумя дискретными положениями
{ S7_Optimized_Access := 'FALSE' }
VERSION : 0.1
// stored: AutoNumber false, IsIECCheckEnabled false, SetENOAutomatically false, UDAEnableTagReadback false
   VAR_INPUT
      All_Block : Bool;   // Аварийный останов
   END_VAR
   VAR_IN_OUT
      FB_QF : Bool;   // защитный автомат / Защитный автомат
      FB_KM_Open : Bool;   // Пускатель - открыть
      FB_KM_Close : Bool;   // Пускатель - закрыть
      FB_Open : Bool;   // ОС - открыто
      FB_Close : Bool;   // ОС - закрыто
      S_Alarm : Bool;   // Наличие аварии
      CMD_Open : Bool;   // Команда - открыть
      CMD_Close : Bool;   // Команда - закрыть
   END_VAR
   VAR DB_SPECIFIC
      CMD : "CMD";   // Основные команды / Блок команд
      Mode : Int;   // Режим работы
      Status : Int;   // Статус устройства
      Use : Struct   // Функционал
         QF { S7_SetPoint := 'True'} : Bool;   // Защитный автомат
         KM_Open { S7_SetPoint := 'True'} : Bool;   // Пускатель - открыть
         KM_Close { S7_SetPoint := 'True'} : Bool;   // Пускатель - закрыть
         Open { S7_SetPoint := 'True'} : Bool := true;   // ОС - открыто
         Close { S7_SetPoint := 'True'} : Bool := true;   // ОС - закрыто
         One_KM { S7_SetPoint := 'True'} : Bool;   // Общий пускатель
         Electro { S7_SetPoint := 'True'} : Bool;   // Электропривод (остановка при срабатывании концевика)
         Cross { S7_SetPoint := 'True'} : Bool;   // Кросс-замена датчиков
         CMD_Open { S7_SetPoint := 'True'} : Bool := true;
         CMD_Close { S7_SetPoint := 'True'} : Bool;
         CMD_Reset : Bool;
         Local_Keys { S7_SetPoint := 'True'} : Bool;
         Local_EndPoint : Bool := true;
      END_STRUCT;
      FB : Struct   // Функционал
         QF : Bool;   // Защитный автомат
         KM_Open : Bool;   // Пускатель - открыть
         KM_Close : Bool;   // Пускатель - закрыть
         Open : Bool;   // ОС - открыто
         Close : Bool;   // ОС - закрыто
         Reserv : Bool;
         Local_Open : Bool;   // Локальное открытие
         Local_Close : Bool;   // Локальное закрытие
      END_STRUCT;
      ON : Bool;   // Успешно запущено
      OFF : Bool;   // Успешно остановлено
      REQ_Open : Bool;   // Запрос на открытие
      REQ_Close : Bool;   // Запрос на закрытие
   END_VAR
   VAR
      Tx { S7_SetPoint := 'True'} : Array[0..4] of "Time_S";   // Блок таймеров
   END_VAR
   VAR DB_SPECIFIC
      Inv : Struct   // Инверсия сигналов
         CMD { S7_SetPoint := 'True'} : Bool;   // Команда запуска
         QF { S7_SetPoint := 'True'} : Bool;   // Защитный автомат
         KM_Open { S7_SetPoint := 'True'} : Bool;   // Пускатель - открыть
         KM_Close { S7_SetPoint := 'True'} : Bool;   // Пускатель - закрыть
         Serivce { S7_SetPoint := 'True'} : Bool;   // Сервисный выключатель
         Open { S7_SetPoint := 'True'} : Bool;   // ОС - открыто
         Close { S7_SetPoint := 'True'} : Bool;   // ОС - закрыто
         Local_Open { S7_SetPoint := 'True'} : Bool;   // Локальное открытие
         Local_Close { S7_SetPoint := 'True'} : Bool;   // Локальное закрытие
      END_STRUCT;
      Alarm : Struct   // Сбор аварий / Список аварий
         Block : Bool;   // Аварийная остановка
         QF : Bool;   // привод не готов / Выбило защитный автомат
         KM_Open : Bool;   // Не сработал пускатель - открыть
         KM_Close : Bool;   // Не сработал пускатель - закрыть
         Two_S : Bool;   // Две ОС
         Open : Bool;   // Не сработал концевик - открыто
         Close : Bool;   // термозащита / Не сработал концевик - закрыто
         OpTime : Bool;
      END_STRUCT;
      Alarms : Word;   // Слово аварий
      Events : Word;
      pos : Array[0..15] of Bool;
      OpTime_h : DInt;   // наработка (ч)
      OpTime_s { S7_SetPoint := 'True'} : DInt;   // наработка (с)
      CodeID { S7_SetPoint := 'True'} : Int;   // Код датчика для привязки в скаде
      Indirect : Struct
         FB_QF { S7_SetPoint := 'True'} : Bool := true;   // защитный автомат / Защитный автомат
         FB_KM_Open { S7_SetPoint := 'True'} : Bool := true;   // Пускатель - открыть
         FB_KM_Close { S7_SetPoint := 'True'} : Bool := true;   // Пускатель - закрыть
         FB_Open { S7_SetPoint := 'True'} : Bool := true;   // ОС - открыто
         FB_Close { S7_SetPoint := 'True'} : Bool := true;   // ОС - закрыто
         CMD_Open { S7_SetPoint := 'True'} : Bool := true;   // Команда на открытие
         CMD_Close { S7_SetPoint := 'True'} : Bool := true;   // Команда на закрытие
      END_STRUCT;
      Indirect_BYTE : Struct
         FB_QF { S7_SetPoint := 'True'} : Int;   // защитный автомат / Защитный автомат
         FB_KM_Open { S7_SetPoint := 'True'} : Int;   // Пускатель - открыть
         FB_KM_Close { S7_SetPoint := 'True'} : Int;   // Пускатель - закрыть
         FB_Open { S7_SetPoint := 'True'} : Int;   // ОС - открыто
         FB_Close { S7_SetPoint := 'True'} : Int;   // ОС - закрыто
         CMD_Open { S7_SetPoint := 'True'} : Int;   // Команда на открытие
         CMD_Close { S7_SetPoint := 'True'} : Int;   // Команда на закрытие
         CMD_Reset : Int;
      END_STRUCT;
      Indirect_BIT : Struct
         FB_QF { S7_SetPoint := 'True'} : Int := 9;   // защитный автомат / Защитный автомат
         FB_KM_Open { S7_SetPoint := 'True'} : Int := 9;   // Пускатель - открыть
         FB_KM_Close { S7_SetPoint := 'True'} : Int := 9;   // Пускатель - закрыть
         FB_Open { S7_SetPoint := 'True'} : Int := 9;   // ОС - открыто
         FB_Close { S7_SetPoint := 'True'} : Int := 9;   // ОС - закрыто
         CMD_Open { S7_SetPoint := 'True'} : Int := 9;   // Команда на открытие
         CMD_Close { S7_SetPoint := 'True'} : Int := 9;   // Команда на закрытие
         CMD_Reset : Int;
      END_STRUCT;
   END_VAR
   VAR_TEMP
      ev : Bool;
      xQF : Bool;
      xKM_Open : Bool;
      xKM_Close : Bool;
      xOpen : Bool;
      xClose : Bool;
   END_VAR
   VAR_TEMP   // added for the SCL form of the ladder/FBD networks
      _w1 : Bool;
      _w2 : Bool;
      _w3 : Bool;
      _w4 : Bool;
      _w5 : Bool;
      _w6 : Bool;
      _w7 : Bool;
      _w8 : Bool;
      _w9 : Bool;
      _w10 : Bool;
      _w11 : Bool;
      _w12 : Bool;
      _w13 : Bool;
      _w14 : Bool;
      _w15 : Bool;
      _w16 : Bool;
      _w17 : Bool;
      _w18 : Bool;
      _w19 : Bool;
      _w20 : Bool;
      _w21 : Bool;
      _w22 : Bool;
      _w23 : Bool;
      _w24 : Bool;
      _w25 : Bool;
      _w26 : Bool;
   END_VAR
BEGIN

REGION Network 1: Режим глобальной симуляции
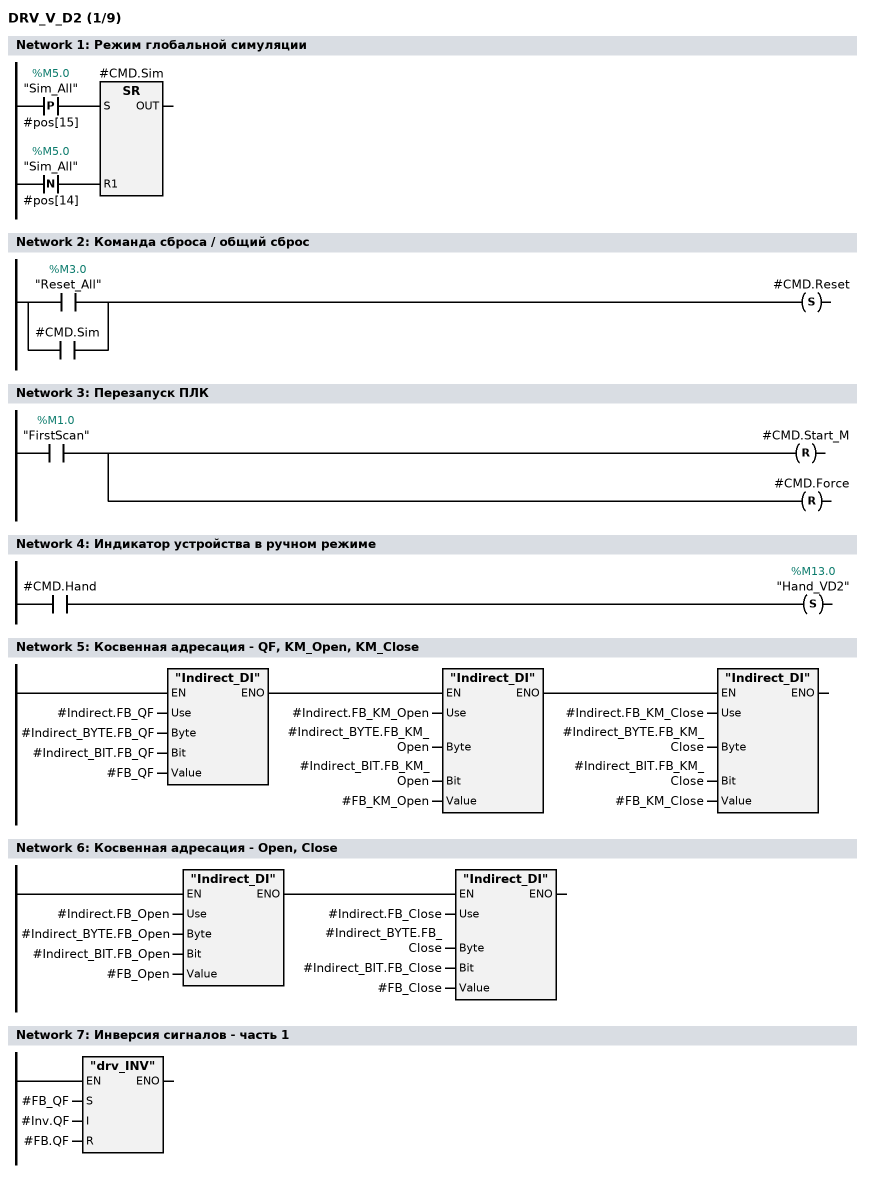
   RUNG wire#powerrail
      P_Contact(operand := "Sim_All", bit := #pos[15])
      S_SR(operand := #CMD.Sim, r1 := wire#w1)
   END_RUNG
   RUNG wire#powerrail
      N_Contact(operand := "Sim_All", bit := #pos[14])
   END_RUNG wire#w1
   // the same network as SCL:
   #_w1 := "Sim_All" AND NOT #pos[15];   // rising edge of "Sim_All"
   #pos[15] := "Sim_All";
   #_w2 := NOT "Sim_All" AND #pos[14];   // falling edge of "Sim_All"
   #pos[14] := "Sim_All";
   IF #_w1 THEN
       #CMD.Sim := TRUE;   // SR flip-flop
   END_IF;
   IF #_w2 THEN #CMD.Sim := FALSE; END_IF;
END_REGION

REGION Network 2: Команда сброса / общий сброс
   RUNG wire#powerrail
      Contact( "Reset_All" )
      wire#w1
      S_Coil( #CMD.Reset )
   END_RUNG
   RUNG wire#powerrail
      Contact( #CMD.Sim )
   END_RUNG wire#w1
   // the same network as SCL:
   IF "Reset_All" OR #CMD.Sim THEN #CMD.Reset := TRUE; END_IF;
END_REGION

REGION Network 3: Перезапуск ПЛК
   RUNG wire#powerrail
      Contact( "FirstScan" )
      wire#w1
      R_Coil( #CMD.Start_M )
   END_RUNG
   RUNG wire#w1
      R_Coil( #CMD.Force )
   END_RUNG
   // the same network as SCL:
   IF "FirstScan" THEN
       #CMD.Start_M := FALSE;
       #CMD.Force := FALSE;
   END_IF;
END_REGION

REGION Network 4: Индикатор устройства в ручном режиме
   RUNG wire#powerrail
      Contact( #CMD.Hand )
      S_Coil( "Hand_VD2" )
   END_RUNG
   // the same network as SCL:
   IF #CMD.Hand THEN "Hand_VD2" := TRUE; END_IF;
END_REGION

REGION Network 5: Косвенная адресация - QF, KM_Open, KM_Close
   RUNG wire#powerrail
      "Indirect_DI"(Use := #Indirect.FB_QF, "Byte" := #Indirect_BYTE.FB_QF, Bit := #Indirect_BIT.FB_QF, Value := #FB_QF)
      "Indirect_DI"(Use := #Indirect.FB_KM_Open, "Byte" := #Indirect_BYTE.FB_KM_Open, Bit := #Indirect_BIT.FB_KM_Open, Value := #FB_KM_Open)
      "Indirect_DI"(Use := #Indirect.FB_KM_Close, "Byte" := #Indirect_BYTE.FB_KM_Close, Bit := #Indirect_BIT.FB_KM_Close, Value := #FB_KM_Close)
   END_RUNG
   // the same network as SCL:
   "Indirect_DI"(Use := #Indirect.FB_QF,
                 "Byte" := #Indirect_BYTE.FB_QF,
                 Bit := #Indirect_BIT.FB_QF,
                 Value := #FB_QF,
                 ENO => #_w1);
   "Indirect_DI"(EN := #_w1,
                 Use := #Indirect.FB_KM_Open,
                 "Byte" := #Indirect_BYTE.FB_KM_Open,
                 Bit := #Indirect_BIT.FB_KM_Open,
                 Value := #FB_KM_Open,
                 ENO => #_w2);
   IF #_w2 THEN
       "Indirect_DI"(Use := #Indirect.FB_KM_Close,
                     "Byte" := #Indirect_BYTE.FB_KM_Close,
                     Bit := #Indirect_BIT.FB_KM_Close,
                     Value := #FB_KM_Close);
   END_IF;
END_REGION

REGION Network 6: Косвенная адресация - Open, Close
   RUNG wire#powerrail
      "Indirect_DI"(Use := #Indirect.FB_Open, "Byte" := #Indirect_BYTE.FB_Open, Bit := #Indirect_BIT.FB_Open, Value := #FB_Open)
      "Indirect_DI"(Use := #Indirect.FB_Close, "Byte" := #Indirect_BYTE.FB_Close, Bit := #Indirect_BIT.FB_Close, Value := #FB_Close)
   END_RUNG
   // the same network as SCL:
   "Indirect_DI"(Use := #Indirect.FB_Open,
                 "Byte" := #Indirect_BYTE.FB_Open,
                 Bit := #Indirect_BIT.FB_Open,
                 Value := #FB_Open,
                 ENO => #_w1);
   IF #_w1 THEN
       "Indirect_DI"(Use := #Indirect.FB_Close,
                     "Byte" := #Indirect_BYTE.FB_Close,
                     Bit := #Indirect_BIT.FB_Close,
                     Value := #FB_Close);
   END_IF;
END_REGION

REGION Network 7: Инверсия сигналов - часть 1
   RUNG wire#powerrail
      "drv_INV"(S := #FB_QF, I := #Inv.QF, R := #FB.QF)
   END_RUNG
   // the same network as SCL:
   "drv_INV"(S := #FB_QF, I := #Inv.QF, R := #FB.QF);
END_REGION

REGION Network 8: ОС
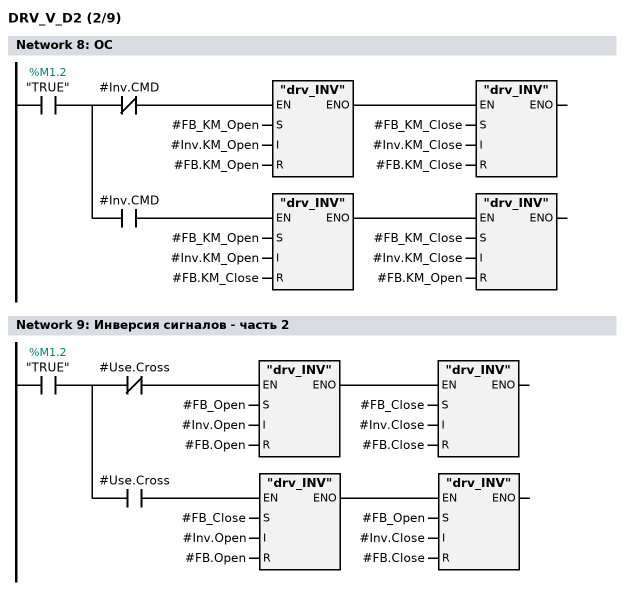
   RUNG wire#powerrail
      Contact( "TRUE" )
      wire#w1
      I_Contact( #Inv.CMD )
      "drv_INV"(S := #FB_KM_Open, I := #Inv.KM_Open, R := #FB.KM_Open)
      "drv_INV"(S := #FB_KM_Close, I := #Inv.KM_Close, R := #FB.KM_Close)
   END_RUNG
   RUNG wire#w1
      Contact( #Inv.CMD )
      "drv_INV"(S := #FB_KM_Open, I := #Inv.KM_Open, R := #FB.KM_Close)
      "drv_INV"(S := #FB_KM_Close, I := #Inv.KM_Close, R := #FB.KM_Open)
   END_RUNG
   // the same network as SCL:
   #_w2 := "TRUE";
   "drv_INV"(EN := "TRUE" AND NOT #Inv.CMD, S := #FB_KM_Open, I := #Inv.KM_Open, R := #FB.KM_Open, ENO => #_w1);
   IF #_w1 THEN "drv_INV"(S := #FB_KM_Close, I := #Inv.KM_Close, R := #FB.KM_Close); END_IF;
   "drv_INV"(EN := #_w2 AND #Inv.CMD, S := #FB_KM_Open, I := #Inv.KM_Open, R := #FB.KM_Close, ENO => #_w3);
   IF #_w3 THEN "drv_INV"(S := #FB_KM_Close, I := #Inv.KM_Close, R := #FB.KM_Open); END_IF;
END_REGION

REGION Network 9: Инверсия сигналов - часть 2
   RUNG wire#powerrail
      Contact( "TRUE" )
      wire#w1
      I_Contact( #Use.Cross )
      "drv_INV"(S := #FB_Open, I := #Inv.Open, R := #FB.Open)
      "drv_INV"(S := #FB_Close, I := #Inv.Close, R := #FB.Close)
   END_RUNG
   RUNG wire#w1
      Contact( #Use.Cross )
      "drv_INV"(S := #FB_Close, I := #Inv.Open, R := #FB.Open)
      "drv_INV"(S := #FB_Open, I := #Inv.Close, R := #FB.Close)
   END_RUNG
   // the same network as SCL:
   #_w2 := "TRUE";
   "drv_INV"(EN := "TRUE" AND NOT #Use.Cross, S := #FB_Open, I := #Inv.Open, R := #FB.Open, ENO => #_w1);
   IF #_w1 THEN "drv_INV"(S := #FB_Close, I := #Inv.Close, R := #FB.Close); END_IF;
   "drv_INV"(EN := #_w2 AND #Use.Cross, S := #FB_Close, I := #Inv.Open, R := #FB.Open, ENO => #_w3);
   IF #_w3 THEN "drv_INV"(S := #FB_Open, I := #Inv.Close, R := #FB.Close); END_IF;
END_REGION

REGION Network 10: Заглушка индикаторов ОС
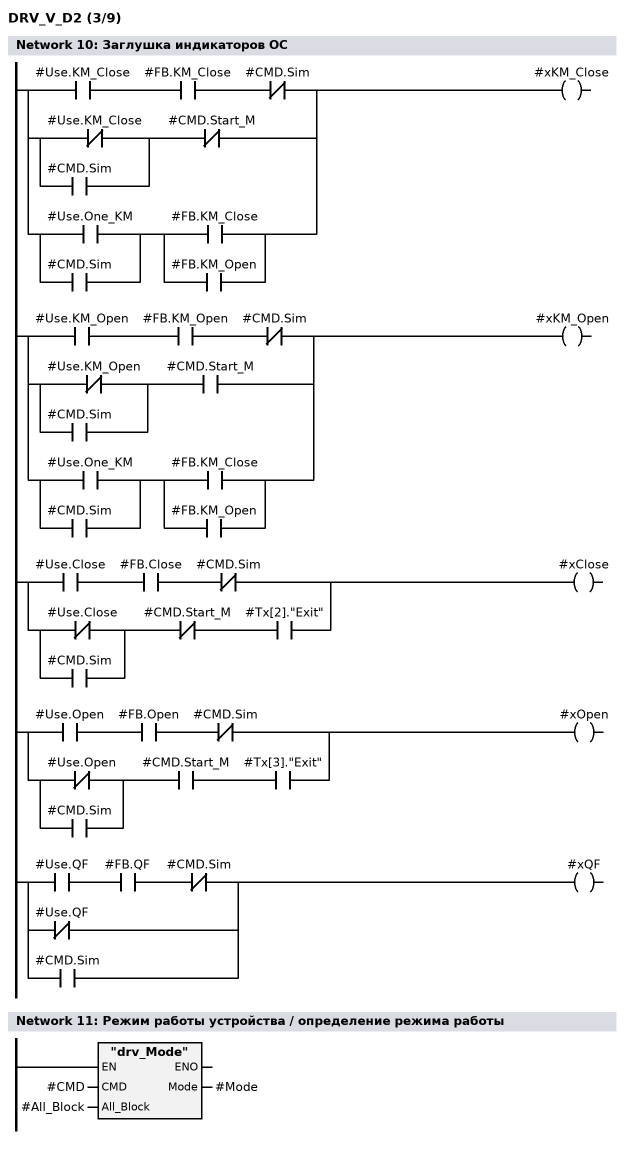
   RUNG wire#powerrail
      Contact( #Use.KM_Close )
      Contact( #FB.KM_Close )
      I_Contact( #CMD.Sim )
      wire#w1
      Coil( #xKM_Close )
   END_RUNG
   RUNG wire#powerrail
      I_Contact( #Use.KM_Close )
      wire#w2
      I_Contact( #CMD.Start_M )
   END_RUNG wire#w1
   RUNG wire#powerrail
      Contact( #CMD.Sim )
   END_RUNG wire#w2
   RUNG wire#powerrail
      Contact( #Use.One_KM )
      wire#w3
      Contact( #FB.KM_Close )
   END_RUNG wire#w1
   RUNG wire#powerrail
      Contact( #CMD.Sim )
   END_RUNG wire#w3
   RUNG wire#w3
      Contact( #FB.KM_Open )
   END_RUNG wire#w1
   RUNG wire#powerrail
      Contact( #Use.KM_Open )
      Contact( #FB.KM_Open )
      I_Contact( #CMD.Sim )
      wire#w4
      Coil( #xKM_Open )
   END_RUNG
   RUNG wire#powerrail
      I_Contact( #Use.KM_Open )
      wire#w5
      Contact( #CMD.Start_M )
   END_RUNG wire#w4
   RUNG wire#powerrail
      Contact( #CMD.Sim )
   END_RUNG wire#w5
   RUNG wire#powerrail
      Contact( #Use.One_KM )
      wire#w6
      Contact( #FB.KM_Close )
   END_RUNG wire#w4
   RUNG wire#powerrail
      Contact( #CMD.Sim )
   END_RUNG wire#w6
   RUNG wire#w6
      Contact( #FB.KM_Open )
   END_RUNG wire#w4
   RUNG wire#powerrail
      Contact( #Use.Close )
      Contact( #FB.Close )
      I_Contact( #CMD.Sim )
      wire#w7
      Coil( #xClose )
   END_RUNG
   RUNG wire#powerrail
      I_Contact( #Use.Close )
      wire#w8
      I_Contact( #CMD.Start_M )
      Contact( #Tx[2]."Exit" )
   END_RUNG wire#w7
   RUNG wire#powerrail
      Contact( #CMD.Sim )
   END_RUNG wire#w8
   RUNG wire#powerrail
      Contact( #Use.Open )
      Contact( #FB.Open )
      I_Contact( #CMD.Sim )
      wire#w9
      Coil( #xOpen )
   END_RUNG
   RUNG wire#powerrail
      I_Contact( #Use.Open )
      wire#w10
      Contact( #CMD.Start_M )
      Contact( #Tx[3]."Exit" )
   END_RUNG wire#w9
   RUNG wire#powerrail
      Contact( #CMD.Sim )
   END_RUNG wire#w10
   RUNG wire#powerrail
      Contact( #Use.QF )
      Contact( #FB.QF )
      I_Contact( #CMD.Sim )
      wire#w11
      Coil( #xQF )
   END_RUNG
   RUNG wire#powerrail
      I_Contact( #Use.QF )
   END_RUNG wire#w11
   RUNG wire#powerrail
      Contact( #CMD.Sim )
   END_RUNG wire#w11
   // the same network as SCL:
   #xKM_Close := (#Use.KM_Close AND #FB.KM_Close AND NOT #CMD.Sim) OR ((NOT #Use.KM_Close OR #CMD.Sim) AND NOT #CMD.Start_M) OR ((#Use.One_KM OR #CMD.Sim) AND (#FB.KM_Close OR #FB.KM_Open));
   #xKM_Open := (#Use.KM_Open AND #FB.KM_Open AND NOT #CMD.Sim) OR ((NOT #Use.KM_Open OR #CMD.Sim) AND #CMD.Start_M) OR ((#Use.One_KM OR #CMD.Sim) AND (#FB.KM_Close OR #FB.KM_Open));
   #xClose := (#Use.Close AND #FB.Close AND NOT #CMD.Sim) OR ((NOT #Use.Close OR #CMD.Sim) AND NOT #CMD.Start_M AND #Tx[2]."Exit");
   #xOpen := (#Use.Open AND #FB.Open AND NOT #CMD.Sim) OR ((NOT #Use.Open OR #CMD.Sim) AND #CMD.Start_M AND #Tx[3]."Exit");
   #xQF := (#Use.QF AND #FB.QF AND NOT #CMD.Sim) OR NOT #Use.QF OR #CMD.Sim;
END_REGION

REGION Network 11: Режим работы устройства / определение режима работы
   RUNG wire#powerrail
      "drv_Mode"(CMD := #CMD, All_Block := #All_Block, Mode => #Mode)
   END_RUNG
   // the same network as SCL:
   "drv_Mode"(CMD := #CMD, All_Block := #All_Block, Mode => #Mode);
END_REGION

REGION Network 12: Управление запуском
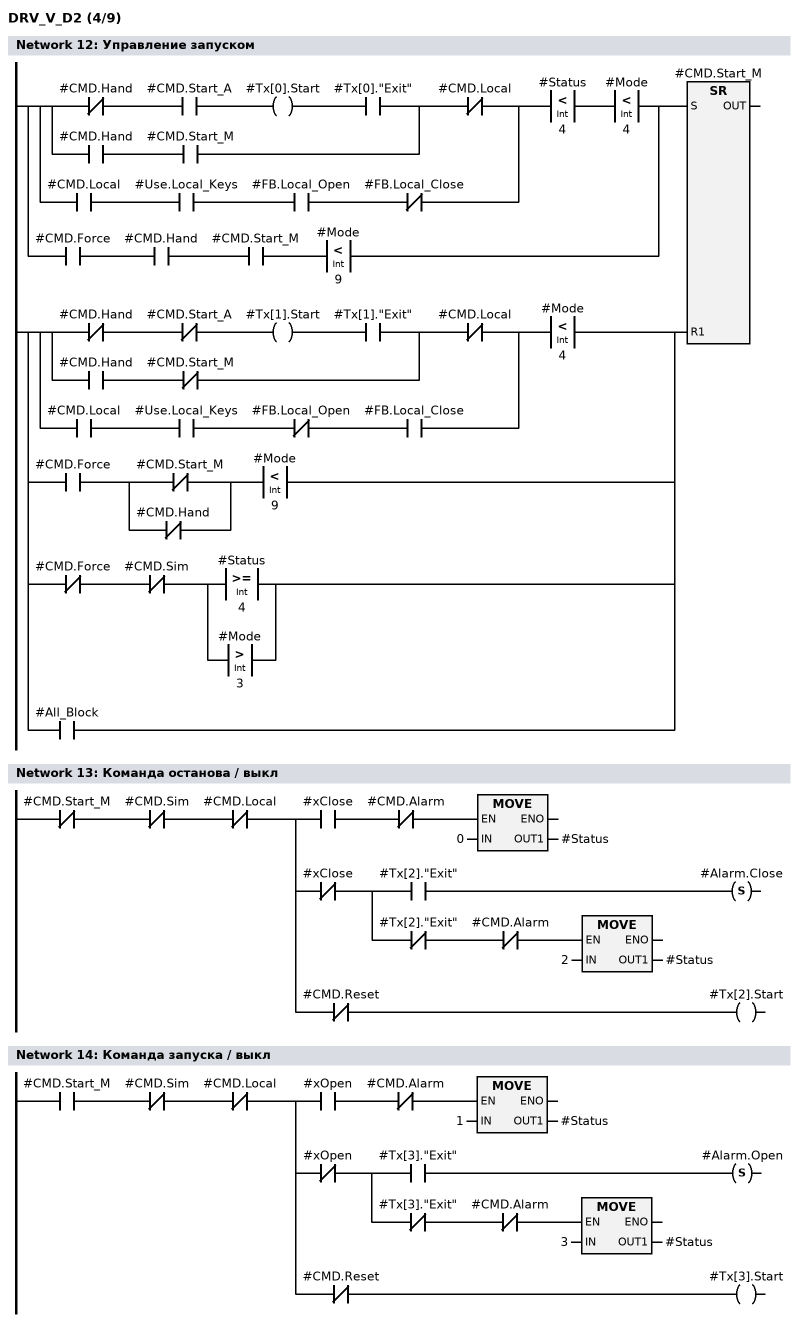
   RUNG wire#powerrail
      I_Contact( #CMD.Hand )
      Contact( #CMD.Start_A )
      Coil( #Tx[0].Start )
      Contact( #Tx[0]."Exit" )
      wire#w1
      I_Contact( #CMD.Local )
      wire#w2
      { S7_Templates := "SrcType := Int" } LT_Contact(in1 := #Status, in2 := 4)
      { S7_Templates := "SrcType := Int" } LT_Contact(in1 := #Mode, in2 := 4)
      wire#w3
      S_SR(operand := #CMD.Start_M, r1 := wire#w9)
   END_RUNG
   RUNG wire#powerrail
      Contact( #CMD.Hand )
      Contact( #CMD.Start_M )
   END_RUNG wire#w1
   RUNG wire#powerrail
      Contact( #CMD.Local )
      Contact( #Use.Local_Keys )
      Contact( #FB.Local_Open )
      I_Contact( #FB.Local_Close )
   END_RUNG wire#w2
   RUNG wire#powerrail
      Contact( #CMD.Force )
      Contact( #CMD.Hand )
      Contact( #CMD.Start_M )
      { S7_Templates := "SrcType := Int" } LT_Contact(in1 := #Mode, in2 := 9)
   END_RUNG wire#w3
   RUNG wire#powerrail
      I_Contact( #CMD.Hand )
      I_Contact( #CMD.Start_A )
      Coil( #Tx[1].Start )
      Contact( #Tx[1]."Exit" )
      wire#w4
      I_Contact( #CMD.Local )
      wire#w5
      { S7_Templates := "SrcType := Int" } LT_Contact(in1 := #Mode, in2 := 4)
   END_RUNG wire#w9
   RUNG wire#powerrail
      Contact( #CMD.Hand )
      I_Contact( #CMD.Start_M )
   END_RUNG wire#w4
   RUNG wire#powerrail
      Contact( #CMD.Local )
      Contact( #Use.Local_Keys )
      I_Contact( #FB.Local_Open )
      Contact( #FB.Local_Close )
   END_RUNG wire#w5
   RUNG wire#powerrail
      Contact( #CMD.Force )
      wire#w6
      I_Contact( #CMD.Start_M )
      wire#w7
      { S7_Templates := "SrcType := Int" } LT_Contact(in1 := #Mode, in2 := 9)
   END_RUNG wire#w9
   RUNG wire#w6
      I_Contact( #CMD.Hand )
   END_RUNG wire#w7
   RUNG wire#powerrail
      I_Contact( #CMD.Force )
      I_Contact( #CMD.Sim )
      wire#w8
      { S7_Templates := "SrcType := Int" } GE_Contact(in1 := #Status, in2 := 4)
   END_RUNG wire#w9
   RUNG wire#w8
      { S7_Templates := "SrcType := Int" } GT_Contact(in1 := #Mode, in2 := 3)
   END_RUNG wire#w9
   RUNG wire#powerrail
      Contact( #All_Block )
   END_RUNG wire#w9
   // the same network as SCL:
   #Tx[0].Start := NOT #CMD.Hand AND #CMD.Start_A;
   #_w1 := (((((NOT #CMD.Hand AND #CMD.Start_A AND #Tx[0]."Exit") OR (#CMD.Hand AND #CMD.Start_M)) AND NOT #CMD.Local) OR (#CMD.Local AND #Use.Local_Keys AND #FB.Local_Open AND NOT #FB.Local_Close)) AND (#Status < 4) AND (#Mode < 4)) OR (#CMD.Force AND #CMD.Hand AND #CMD.Start_M AND (#Mode < 9));
   #Tx[1].Start := NOT #CMD.Hand AND NOT #CMD.Start_A;
   #_w2 := (((((NOT #CMD.Hand AND NOT #CMD.Start_A AND #Tx[1]."Exit") OR (#CMD.Hand AND NOT #CMD.Start_M)) AND NOT #CMD.Local) OR (#CMD.Local AND #Use.Local_Keys AND NOT #FB.Local_Open AND #FB.Local_Close)) AND (#Mode < 4)) OR (#CMD.Force AND (NOT #CMD.Start_M OR NOT #CMD.Hand) AND (#Mode < 9)) OR (NOT #CMD.Force AND NOT #CMD.Sim AND ((#Status >= 4) OR (#Mode > 3))) OR #All_Block;
   IF #_w1 THEN
       #CMD.Start_M := TRUE;   // SR flip-flop
   END_IF;
   IF #_w2 THEN #CMD.Start_M := FALSE; END_IF;
END_REGION

REGION Network 13: Команда останова / выкл
   RUNG wire#powerrail
      I_Contact( #CMD.Start_M )
      I_Contact( #CMD.Sim )
      I_Contact( #CMD.Local )
      wire#w1
      Contact( #xClose )
      I_Contact( #CMD.Alarm )
      { S7_GenerateENO := "TRUE" } Move(in := 0, out1 => #Status)
   END_RUNG
   RUNG wire#w1
      I_Contact( #xClose )
      wire#w2
      Contact( #Tx[2]."Exit" )
      S_Coil( #Alarm.Close )
   END_RUNG
   RUNG wire#w2
      I_Contact( #Tx[2]."Exit" )
      I_Contact( #CMD.Alarm )
      { S7_GenerateENO := "TRUE" } Move(in := 2, out1 => #Status)
   END_RUNG
   RUNG wire#w1
      I_Contact( #CMD.Reset )
      Coil( #Tx[2].Start )
   END_RUNG
   // the same network as SCL:
   #_w1 := NOT #CMD.Start_M AND NOT #CMD.Sim AND NOT #CMD.Local;
   IF #_w1 AND #xClose AND NOT #CMD.Alarm THEN #Status := 0; END_IF;
   #_w2 := #_w1 AND NOT #xClose;
   IF #_w2 AND #Tx[2]."Exit" THEN #Alarm.Close := TRUE; END_IF;
   IF #_w2 AND NOT #Tx[2]."Exit" AND NOT #CMD.Alarm THEN #Status := 2; END_IF;
   #Tx[2].Start := #_w1 AND NOT #CMD.Reset;
END_REGION

REGION Network 14: Команда запуска / выкл
   RUNG wire#powerrail
      Contact( #CMD.Start_M )
      I_Contact( #CMD.Sim )
      I_Contact( #CMD.Local )
      wire#w1
      Contact( #xOpen )
      I_Contact( #CMD.Alarm )
      { S7_GenerateENO := "TRUE" } Move(in := 1, out1 => #Status)
   END_RUNG
   RUNG wire#w1
      I_Contact( #xOpen )
      wire#w2
      Contact( #Tx[3]."Exit" )
      S_Coil( #Alarm.Open )
   END_RUNG
   RUNG wire#w2
      I_Contact( #Tx[3]."Exit" )
      I_Contact( #CMD.Alarm )
      { S7_GenerateENO := "TRUE" } Move(in := 3, out1 => #Status)
   END_RUNG
   RUNG wire#w1
      I_Contact( #CMD.Reset )
      Coil( #Tx[3].Start )
   END_RUNG
   // the same network as SCL:
   #_w1 := #CMD.Start_M AND NOT #CMD.Sim AND NOT #CMD.Local;
   IF #_w1 AND #xOpen AND NOT #CMD.Alarm THEN #Status := 1; END_IF;
   #_w2 := #_w1 AND NOT #xOpen;
   IF #_w2 AND #Tx[3]."Exit" THEN #Alarm.Open := TRUE; END_IF;
   IF #_w2 AND NOT #Tx[3]."Exit" AND NOT #CMD.Alarm THEN #Status := 3; END_IF;
   #Tx[3].Start := #_w1 AND NOT #CMD.Reset;
END_REGION

REGION Network 15: Режим симуляции
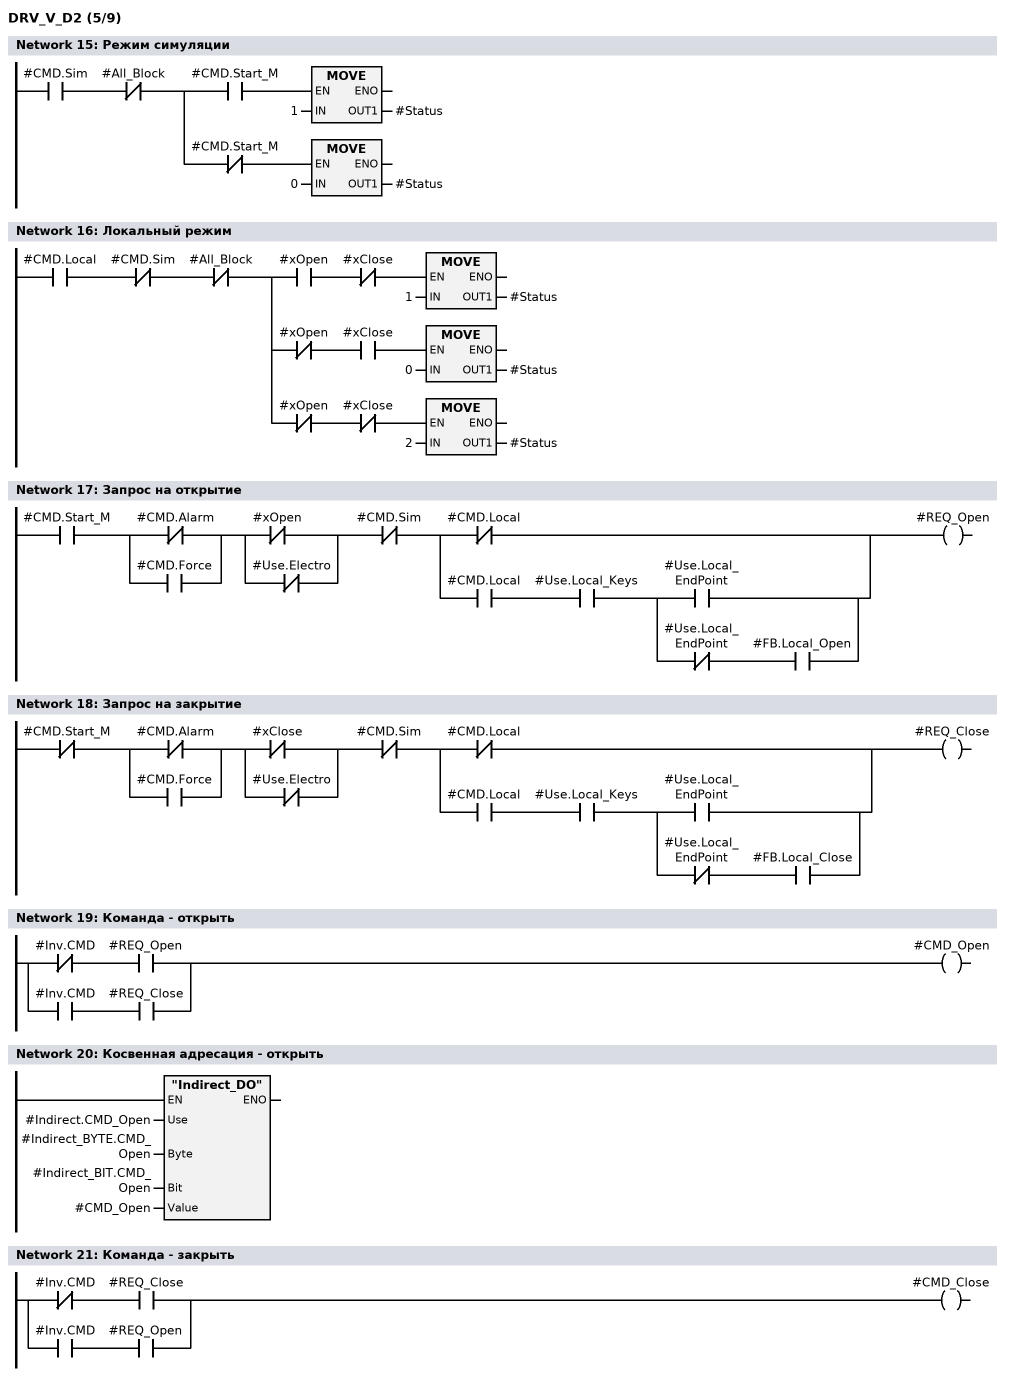
   RUNG wire#powerrail
      Contact( #CMD.Sim )
      I_Contact( #All_Block )
      wire#w1
      Contact( #CMD.Start_M )
      { S7_GenerateENO := "TRUE" } Move(in := 1, out1 => #Status)
   END_RUNG
   RUNG wire#w1
      I_Contact( #CMD.Start_M )
      { S7_GenerateENO := "TRUE" } Move(in := 0, out1 => #Status)
   END_RUNG
   // the same network as SCL:
   #_w1 := #CMD.Sim AND NOT #All_Block;
   IF #_w1 AND #CMD.Start_M THEN #Status := 1; END_IF;
   IF #_w1 AND NOT #CMD.Start_M THEN #Status := 0; END_IF;
END_REGION

REGION Network 16: Локальный режим
   RUNG wire#powerrail
      Contact( #CMD.Local )
      I_Contact( #CMD.Sim )
      I_Contact( #All_Block )
      wire#w1
      Contact( #xOpen )
      I_Contact( #xClose )
      { S7_GenerateENO := "TRUE" } Move(in := 1, out1 => #Status)
   END_RUNG
   RUNG wire#w1
      I_Contact( #xOpen )
      Contact( #xClose )
      { S7_GenerateENO := "TRUE" } Move(in := 0, out1 => #Status)
   END_RUNG
   RUNG wire#w1
      I_Contact( #xOpen )
      I_Contact( #xClose )
      { S7_GenerateENO := "TRUE" } Move(in := 2, out1 => #Status)
   END_RUNG
   // the same network as SCL:
   #_w1 := #CMD.Local AND NOT #CMD.Sim AND NOT #All_Block;
   IF #_w1 AND #xOpen AND NOT #xClose THEN #Status := 1; END_IF;
   IF #_w1 AND NOT #xOpen AND #xClose THEN #Status := 0; END_IF;
   IF #_w1 AND NOT #xOpen AND NOT #xClose THEN #Status := 2; END_IF;
END_REGION

REGION Network 17: Запрос на открытие
   RUNG wire#powerrail
      Contact( #CMD.Start_M )
      wire#w1
      I_Contact( #CMD.Alarm )
      wire#w2
      I_Contact( #xOpen )
      wire#w3
      I_Contact( #CMD.Sim )
      wire#w4
      I_Contact( #CMD.Local )
      wire#w5
      Coil( #REQ_Open )
   END_RUNG
   RUNG wire#w1
      Contact( #CMD.Force )
   END_RUNG wire#w2
   RUNG wire#w2
      I_Contact( #Use.Electro )
   END_RUNG wire#w3
   RUNG wire#w4
      Contact( #CMD.Local )
      Contact( #Use.Local_Keys )
      wire#w6
      Contact( #Use.Local_EndPoint )
   END_RUNG wire#w5
   RUNG wire#w6
      I_Contact( #Use.Local_EndPoint )
      Contact( #FB.Local_Open )
   END_RUNG wire#w5
   // the same network as SCL:
   #REQ_Open := #CMD.Start_M AND (NOT #CMD.Alarm OR #CMD.Force) AND (NOT #xOpen OR NOT #Use.Electro) AND NOT #CMD.Sim AND (NOT #CMD.Local OR (#CMD.Local AND #Use.Local_Keys AND (#Use.Local_EndPoint OR (NOT #Use.Local_EndPoint AND #FB.Local_Open))));
END_REGION

REGION Network 18: Запрос на закрытие
   RUNG wire#powerrail
      I_Contact( #CMD.Start_M )
      wire#w1
      I_Contact( #CMD.Alarm )
      wire#w2
      I_Contact( #xClose )
      wire#w3
      I_Contact( #CMD.Sim )
      wire#w4
      I_Contact( #CMD.Local )
      wire#w5
      Coil( #REQ_Close )
   END_RUNG
   RUNG wire#w1
      Contact( #CMD.Force )
   END_RUNG wire#w2
   RUNG wire#w2
      I_Contact( #Use.Electro )
   END_RUNG wire#w3
   RUNG wire#w4
      Contact( #CMD.Local )
      Contact( #Use.Local_Keys )
      wire#w6
      Contact( #Use.Local_EndPoint )
   END_RUNG wire#w5
   RUNG wire#w6
      I_Contact( #Use.Local_EndPoint )
      Contact( #FB.Local_Close )
   END_RUNG wire#w5
   // the same network as SCL:
   #REQ_Close := NOT #CMD.Start_M AND (NOT #CMD.Alarm OR #CMD.Force) AND (NOT #xClose OR NOT #Use.Electro) AND NOT #CMD.Sim AND (NOT #CMD.Local OR (#CMD.Local AND #Use.Local_Keys AND (#Use.Local_EndPoint OR (NOT #Use.Local_EndPoint AND #FB.Local_Close))));
END_REGION

REGION Network 19: Команда - открыть
   RUNG wire#powerrail
      I_Contact( #Inv.CMD )
      Contact( #REQ_Open )
      wire#w1
      Coil( #CMD_Open )
   END_RUNG
   RUNG wire#powerrail
      Contact( #Inv.CMD )
      Contact( #REQ_Close )
   END_RUNG wire#w1
   // the same network as SCL:
   #CMD_Open := (NOT #Inv.CMD AND #REQ_Open) OR (#Inv.CMD AND #REQ_Close);
END_REGION

REGION Network 20: Косвенная адресация - открыть
   RUNG wire#powerrail
      "Indirect_DO"(Use := #Indirect.CMD_Open, "Byte" := #Indirect_BYTE.CMD_Open, Bit := #Indirect_BIT.CMD_Open, Value := #CMD_Open)
   END_RUNG
   // the same network as SCL:
   "Indirect_DO"(Use := #Indirect.CMD_Open,
                 "Byte" := #Indirect_BYTE.CMD_Open,
                 Bit := #Indirect_BIT.CMD_Open,
                 Value := #CMD_Open);
END_REGION

REGION Network 21: Команда - закрыть
   RUNG wire#powerrail
      I_Contact( #Inv.CMD )
      Contact( #REQ_Close )
      wire#w1
      Coil( #CMD_Close )
   END_RUNG
   RUNG wire#powerrail
      Contact( #Inv.CMD )
      Contact( #REQ_Open )
   END_RUNG wire#w1
   // the same network as SCL:
   #CMD_Close := (NOT #Inv.CMD AND #REQ_Close) OR (#Inv.CMD AND #REQ_Open);
END_REGION

REGION Network 22: Косвенная адресация - закрыть
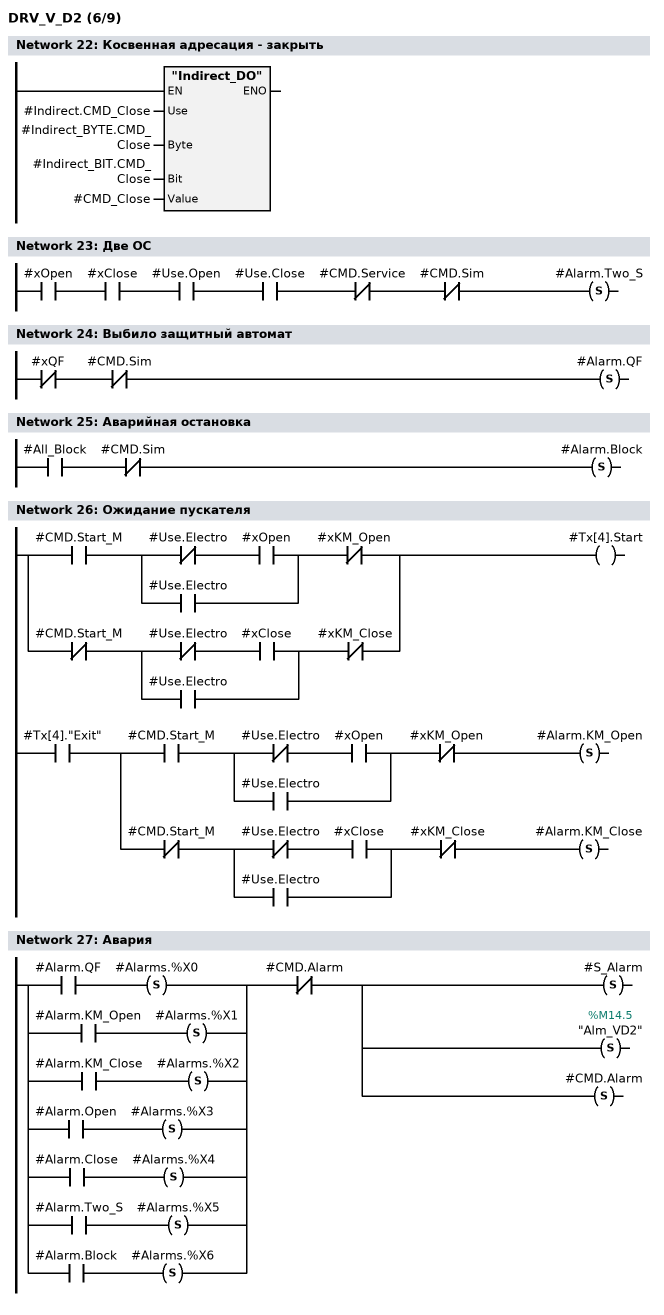
   RUNG wire#powerrail
      "Indirect_DO"(Use := #Indirect.CMD_Close, "Byte" := #Indirect_BYTE.CMD_Close, Bit := #Indirect_BIT.CMD_Close, Value := #CMD_Close)
   END_RUNG
   // the same network as SCL:
   "Indirect_DO"(Use := #Indirect.CMD_Close,
                 "Byte" := #Indirect_BYTE.CMD_Close,
                 Bit := #Indirect_BIT.CMD_Close,
                 Value := #CMD_Close);
END_REGION

REGION Network 23: Две ОС
   RUNG wire#powerrail
      Contact( #xOpen )
      Contact( #xClose )
      Contact( #Use.Open )
      Contact( #Use.Close )
      I_Contact( #CMD.Service )
      I_Contact( #CMD.Sim )
      S_Coil( #Alarm.Two_S )
   END_RUNG
   // the same network as SCL:
   IF #xOpen AND #xClose AND #Use.Open AND #Use.Close AND NOT #CMD.Service AND NOT #CMD.Sim THEN
       #Alarm.Two_S := TRUE;
   END_IF;
END_REGION

REGION Network 24: Выбило защитный автомат
   RUNG wire#powerrail
      I_Contact( #xQF )
      I_Contact( #CMD.Sim )
      S_Coil( #Alarm.QF )
   END_RUNG
   // the same network as SCL:
   IF NOT #xQF AND NOT #CMD.Sim THEN #Alarm.QF := TRUE; END_IF;
END_REGION

REGION Network 25: Аварийная остановка
   RUNG wire#powerrail
      Contact( #All_Block )
      I_Contact( #CMD.Sim )
      S_Coil( #Alarm.Block )
   END_RUNG
   // the same network as SCL:
   IF #All_Block AND NOT #CMD.Sim THEN #Alarm.Block := TRUE; END_IF;
END_REGION

REGION Network 26: Ожидание пускателя
   RUNG wire#powerrail
      Contact( #CMD.Start_M )
      wire#w1
      I_Contact( #Use.Electro )
      Contact( #xOpen )
      wire#w2
      I_Contact( #xKM_Open )
      wire#w3
      Coil( #Tx[4].Start )
   END_RUNG
   RUNG wire#w1
      Contact( #Use.Electro )
   END_RUNG wire#w2
   RUNG wire#powerrail
      I_Contact( #CMD.Start_M )
      wire#w4
      I_Contact( #Use.Electro )
      Contact( #xClose )
      wire#w5
      I_Contact( #xKM_Close )
   END_RUNG wire#w3
   RUNG wire#w4
      Contact( #Use.Electro )
   END_RUNG wire#w5
   RUNG wire#powerrail
      Contact( #Tx[4]."Exit" )
      wire#w6
      Contact( #CMD.Start_M )
      wire#w7
      I_Contact( #Use.Electro )
      Contact( #xOpen )
      wire#w8
      I_Contact( #xKM_Open )
      S_Coil( #Alarm.KM_Open )
   END_RUNG
   RUNG wire#w7
      Contact( #Use.Electro )
   END_RUNG wire#w8
   RUNG wire#w6
      I_Contact( #CMD.Start_M )
      wire#w9
      I_Contact( #Use.Electro )
      Contact( #xClose )
      wire#w10
      I_Contact( #xKM_Close )
      S_Coil( #Alarm.KM_Close )
   END_RUNG
   RUNG wire#w9
      Contact( #Use.Electro )
   END_RUNG wire#w10
   // the same network as SCL:
   #Tx[4].Start := (#CMD.Start_M AND ((NOT #Use.Electro AND #xOpen) OR #Use.Electro) AND NOT #xKM_Open) OR (NOT #CMD.Start_M AND ((NOT #Use.Electro AND #xClose) OR #Use.Electro) AND NOT #xKM_Close);
   IF #Tx[4]."Exit" AND #CMD.Start_M AND ((NOT #Use.Electro AND #xOpen) OR #Use.Electro) AND NOT #xKM_Open THEN
       #Alarm.KM_Open := TRUE;
   END_IF;
   IF #Tx[4]."Exit" AND NOT #CMD.Start_M AND ((NOT #Use.Electro AND #xClose) OR #Use.Electro) AND NOT #xKM_Close THEN
       #Alarm.KM_Close := TRUE;
   END_IF;
END_REGION

REGION Network 27: Авария
   RUNG wire#powerrail
      Contact( #Alarm.QF )
      S_Coil( #Alarms.%X0 )
      wire#w1
      I_Contact( #CMD.Alarm )
      wire#w2
      S_Coil( #S_Alarm )
   END_RUNG
   RUNG wire#powerrail
      Contact( #Alarm.KM_Open )
      S_Coil( #Alarms.%X1 )
   END_RUNG wire#w1
   RUNG wire#powerrail
      Contact( #Alarm.KM_Close )
      S_Coil( #Alarms.%X2 )
   END_RUNG wire#w1
   RUNG wire#powerrail
      Contact( #Alarm.Open )
      S_Coil( #Alarms.%X3 )
   END_RUNG wire#w1
   RUNG wire#powerrail
      Contact( #Alarm.Close )
      S_Coil( #Alarms.%X4 )
   END_RUNG wire#w1
   RUNG wire#powerrail
      Contact( #Alarm.Two_S )
      S_Coil( #Alarms.%X5 )
   END_RUNG wire#w1
   RUNG wire#powerrail
      Contact( #Alarm.Block )
      S_Coil( #Alarms.%X6 )
   END_RUNG wire#w1
   RUNG wire#w2
      S_Coil( "Alm_VD2" )
   END_RUNG
   RUNG wire#w2
      S_Coil( #CMD.Alarm )
   END_RUNG
   // the same network as SCL:
   IF #Alarm.QF THEN #Alarms.%X0 := TRUE; END_IF;
   IF #Alarm.KM_Open THEN #Alarms.%X1 := TRUE; END_IF;
   IF #Alarm.KM_Close THEN #Alarms.%X2 := TRUE; END_IF;
   IF #Alarm.Open THEN #Alarms.%X3 := TRUE; END_IF;
   IF #Alarm.Close THEN #Alarms.%X4 := TRUE; END_IF;
   IF #Alarm.Two_S THEN #Alarms.%X5 := TRUE; END_IF;
   IF #Alarm.Block THEN #Alarms.%X6 := TRUE; END_IF;
   IF (#Alarm.QF OR #Alarm.KM_Open OR #Alarm.KM_Close OR #Alarm.Open OR #Alarm.Close OR #Alarm.Two_S OR #Alarm.Block) AND NOT #CMD.Alarm THEN
       #S_Alarm := TRUE;
       "Alm_VD2" := TRUE;
       #CMD.Alarm := TRUE;
   END_IF;
END_REGION

REGION Network 28: Статусы при аварии
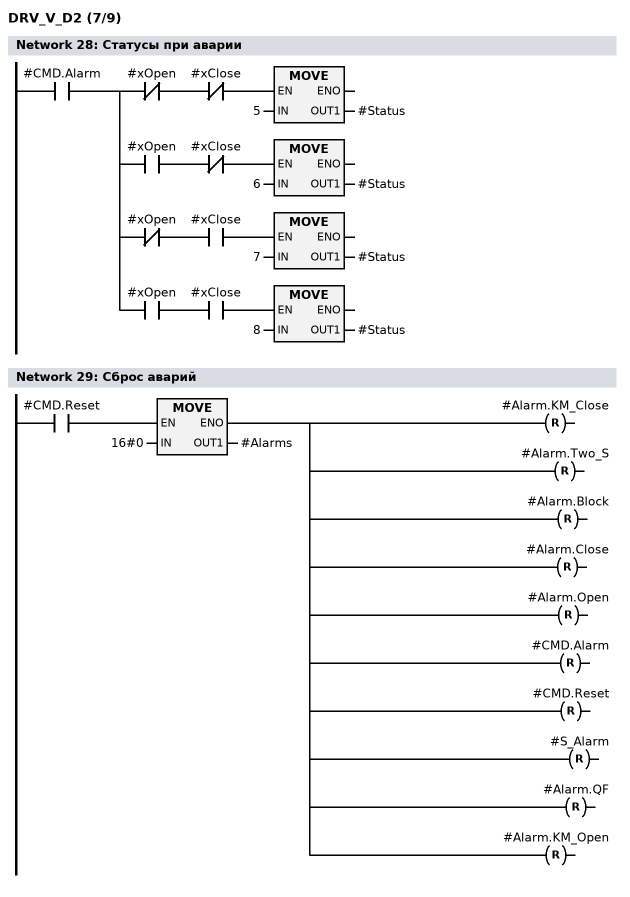
   RUNG wire#powerrail
      Contact( #CMD.Alarm )
      wire#w1
      I_Contact( #xOpen )
      I_Contact( #xClose )
      Move(in := 5, out1 => #Status)
   END_RUNG
   RUNG wire#w1
      Contact( #xOpen )
      I_Contact( #xClose )
      Move(in := 6, out1 => #Status)
   END_RUNG
   RUNG wire#w1
      I_Contact( #xOpen )
      Contact( #xClose )
      Move(in := 7, out1 => #Status)
   END_RUNG
   RUNG wire#w1
      Contact( #xOpen )
      Contact( #xClose )
      Move(in := 8, out1 => #Status)
   END_RUNG
   // the same network as SCL:
   IF #CMD.Alarm AND NOT #xOpen AND NOT #xClose THEN #Status := 5; END_IF;
   IF #CMD.Alarm AND #xOpen AND NOT #xClose THEN #Status := 6; END_IF;
   IF #CMD.Alarm AND NOT #xOpen AND #xClose THEN #Status := 7; END_IF;
   IF #CMD.Alarm AND #xOpen AND #xClose THEN #Status := 8; END_IF;
END_REGION

REGION Network 29: Сброс аварий
   RUNG wire#powerrail
      Contact( #CMD.Reset )
      Move(in := 16#0, out1 => #Alarms)
      wire#w1
      R_Coil( #Alarm.KM_Close )
   END_RUNG
   RUNG wire#w1
      R_Coil( #Alarm.Two_S )
   END_RUNG
   RUNG wire#w1
      R_Coil( #Alarm.Block )
   END_RUNG
   RUNG wire#w1
      R_Coil( #Alarm.Close )
   END_RUNG
   RUNG wire#w1
      R_Coil( #Alarm.Open )
   END_RUNG
   RUNG wire#w1
      R_Coil( #CMD.Alarm )
   END_RUNG
   RUNG wire#w1
      R_Coil( #CMD.Reset )
   END_RUNG
   RUNG wire#w1
      R_Coil( #S_Alarm )
   END_RUNG
   RUNG wire#w1
      R_Coil( #Alarm.QF )
   END_RUNG
   RUNG wire#w1
      R_Coil( #Alarm.KM_Open )
   END_RUNG
   // the same network as SCL:
   IF #CMD.Reset THEN
       #Alarms := 16#0;
       #Alarm.KM_Close := FALSE;
       #Alarm.Two_S := FALSE;
       #Alarm.Block := FALSE;
       #Alarm.Close := FALSE;
       #Alarm.Open := FALSE;
       #CMD.Alarm := FALSE;
   END_IF;
   #_w1 := #CMD.Reset;
   IF #_w1 THEN
       #CMD.Reset := FALSE;
       #S_Alarm := FALSE;
       #Alarm.QF := FALSE;
       #Alarm.KM_Open := FALSE;
   END_IF;
END_REGION

REGION Network 30: События привода
   // 0 - ручной режим активирован
   // 1 - ручной режим деактивирован
   // 2 - принудительный режим активирован
   // 3 - принудительный режим деактивирован
   // 4 - запуск в ручном режиме
   // 5 - останов в ручном режиме
   // 6 - местный режим управления активирован
   // 7 - местный режим управления деактивирован
   // 8 - запущено в местном режиме
   // 9 - остановлено в местном режиме
   // 10 - сервисный режим активирован
   // 11 - сервисный режим деактивирован
   // 12 - проведено сервисное обслуживание
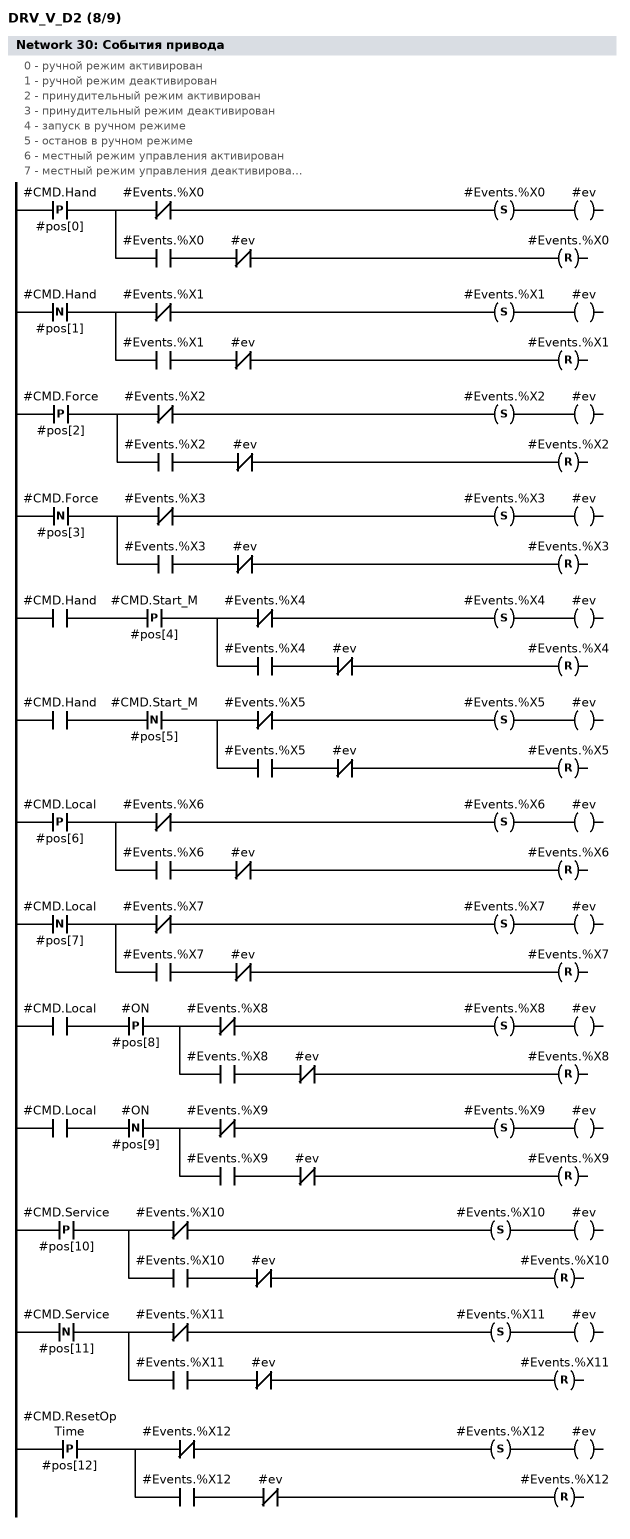
   RUNG wire#powerrail
      P_Contact(operand := #CMD.Hand, bit := #pos[0])
      wire#w1
      I_Contact( #Events.%X0 )
      S_Coil( #Events.%X0 )
      Coil( #ev )
   END_RUNG
   RUNG wire#w1
      Contact( #Events.%X0 )
      I_Contact( #ev )
      R_Coil( #Events.%X0 )
   END_RUNG
   RUNG wire#powerrail
      N_Contact(operand := #CMD.Hand, bit := #pos[1])
      wire#w2
      I_Contact( #Events.%X1 )
      S_Coil( #Events.%X1 )
      Coil( #ev )
   END_RUNG
   RUNG wire#w2
      Contact( #Events.%X1 )
      I_Contact( #ev )
      R_Coil( #Events.%X1 )
   END_RUNG
   RUNG wire#powerrail
      P_Contact(operand := #CMD.Force, bit := #pos[2])
      wire#w3
      I_Contact( #Events.%X2 )
      S_Coil( #Events.%X2 )
      Coil( #ev )
   END_RUNG
   RUNG wire#w3
      Contact( #Events.%X2 )
      I_Contact( #ev )
      R_Coil( #Events.%X2 )
   END_RUNG
   RUNG wire#powerrail
      N_Contact(operand := #CMD.Force, bit := #pos[3])
      wire#w4
      I_Contact( #Events.%X3 )
      S_Coil( #Events.%X3 )
      Coil( #ev )
   END_RUNG
   RUNG wire#w4
      Contact( #Events.%X3 )
      I_Contact( #ev )
      R_Coil( #Events.%X3 )
   END_RUNG
   RUNG wire#powerrail
      Contact( #CMD.Hand )
      P_Contact(operand := #CMD.Start_M, bit := #pos[4])
      wire#w5
      I_Contact( #Events.%X4 )
      S_Coil( #Events.%X4 )
      Coil( #ev )
   END_RUNG
   RUNG wire#w5
      Contact( #Events.%X4 )
      I_Contact( #ev )
      R_Coil( #Events.%X4 )
   END_RUNG
   RUNG wire#powerrail
      Contact( #CMD.Hand )
      N_Contact(operand := #CMD.Start_M, bit := #pos[5])
      wire#w6
      I_Contact( #Events.%X5 )
      S_Coil( #Events.%X5 )
      Coil( #ev )
   END_RUNG
   RUNG wire#w6
      Contact( #Events.%X5 )
      I_Contact( #ev )
      R_Coil( #Events.%X5 )
   END_RUNG
   RUNG wire#powerrail
      P_Contact(operand := #CMD.Local, bit := #pos[6])
      wire#w7
      I_Contact( #Events.%X6 )
      S_Coil( #Events.%X6 )
      Coil( #ev )
   END_RUNG
   RUNG wire#w7
      Contact( #Events.%X6 )
      I_Contact( #ev )
      R_Coil( #Events.%X6 )
   END_RUNG
   RUNG wire#powerrail
      N_Contact(operand := #CMD.Local, bit := #pos[7])
      wire#w8
      I_Contact( #Events.%X7 )
      S_Coil( #Events.%X7 )
      Coil( #ev )
   END_RUNG
   RUNG wire#w8
      Contact( #Events.%X7 )
      I_Contact( #ev )
      R_Coil( #Events.%X7 )
   END_RUNG
   RUNG wire#powerrail
      Contact( #CMD.Local )
      P_Contact(operand := #ON, bit := #pos[8])
      wire#w9
      I_Contact( #Events.%X8 )
      S_Coil( #Events.%X8 )
      Coil( #ev )
   END_RUNG
   RUNG wire#w9
      Contact( #Events.%X8 )
      I_Contact( #ev )
      R_Coil( #Events.%X8 )
   END_RUNG
   RUNG wire#powerrail
      Contact( #CMD.Local )
      N_Contact(operand := #ON, bit := #pos[9])
      wire#w10
      I_Contact( #Events.%X9 )
      S_Coil( #Events.%X9 )
      Coil( #ev )
   END_RUNG
   RUNG wire#w10
      Contact( #Events.%X9 )
      I_Contact( #ev )
      R_Coil( #Events.%X9 )
   END_RUNG
   RUNG wire#powerrail
      P_Contact(operand := #CMD.Service, bit := #pos[10])
      wire#w11
      I_Contact( #Events.%X10 )
      S_Coil( #Events.%X10 )
      Coil( #ev )
   END_RUNG
   RUNG wire#w11
      Contact( #Events.%X10 )
      I_Contact( #ev )
      R_Coil( #Events.%X10 )
   END_RUNG
   RUNG wire#powerrail
      N_Contact(operand := #CMD.Service, bit := #pos[11])
      wire#w12
      I_Contact( #Events.%X11 )
      S_Coil( #Events.%X11 )
      Coil( #ev )
   END_RUNG
   RUNG wire#w12
      Contact( #Events.%X11 )
      I_Contact( #ev )
      R_Coil( #Events.%X11 )
   END_RUNG
   RUNG wire#powerrail
      P_Contact(operand := #CMD.ResetOpTime, bit := #pos[12])
      wire#w13
      I_Contact( #Events.%X12 )
      S_Coil( #Events.%X12 )
      Coil( #ev )
   END_RUNG
   RUNG wire#w13
      Contact( #Events.%X12 )
      I_Contact( #ev )
      R_Coil( #Events.%X12 )
   END_RUNG
   // the same network as SCL:
   #_w1 := #CMD.Hand AND NOT #pos[0];   // rising edge of #CMD.Hand
   #pos[0] := #CMD.Hand;
   #_w2 := #_w1 AND NOT #Events.%X0;
   IF #_w2 THEN #Events.%X0 := TRUE; END_IF;
   #ev := #_w2;
   IF #_w1 AND #Events.%X0 AND NOT #ev THEN #Events.%X0 := FALSE; END_IF;
   #_w3 := NOT #CMD.Hand AND #pos[1];   // falling edge of #CMD.Hand
   #pos[1] := #CMD.Hand;
   #_w4 := #_w3 AND NOT #Events.%X1;
   IF #_w4 THEN #Events.%X1 := TRUE; END_IF;
   #ev := #_w4;
   IF #_w3 AND #Events.%X1 AND NOT #ev THEN #Events.%X1 := FALSE; END_IF;
   #_w5 := #CMD.Force AND NOT #pos[2];   // rising edge of #CMD.Force
   #pos[2] := #CMD.Force;
   #_w6 := #_w5 AND NOT #Events.%X2;
   IF #_w6 THEN #Events.%X2 := TRUE; END_IF;
   #ev := #_w6;
   IF #_w5 AND #Events.%X2 AND NOT #ev THEN #Events.%X2 := FALSE; END_IF;
   #_w7 := NOT #CMD.Force AND #pos[3];   // falling edge of #CMD.Force
   #pos[3] := #CMD.Force;
   #_w8 := #_w7 AND NOT #Events.%X3;
   IF #_w8 THEN #Events.%X3 := TRUE; END_IF;
   #ev := #_w8;
   IF #_w7 AND #Events.%X3 AND NOT #ev THEN #Events.%X3 := FALSE; END_IF;
   #_w9 := #CMD.Hand AND #CMD.Start_M AND NOT #pos[4];   // rising edge of #CMD.Start_M
   #pos[4] := #CMD.Start_M;
   #_w10 := #_w9 AND NOT #Events.%X4;
   IF #_w10 THEN #Events.%X4 := TRUE; END_IF;
   #ev := #_w10;
   IF #_w9 AND #Events.%X4 AND NOT #ev THEN #Events.%X4 := FALSE; END_IF;
   #_w11 := #CMD.Hand AND NOT #CMD.Start_M AND #pos[5];   // falling edge of #CMD.Start_M
   #pos[5] := #CMD.Start_M;
   #_w12 := #_w11 AND NOT #Events.%X5;
   IF #_w12 THEN #Events.%X5 := TRUE; END_IF;
   #ev := #_w12;
   IF #_w11 AND #Events.%X5 AND NOT #ev THEN #Events.%X5 := FALSE; END_IF;
   #_w13 := #CMD.Local AND NOT #pos[6];   // rising edge of #CMD.Local
   #pos[6] := #CMD.Local;
   #_w14 := #_w13 AND NOT #Events.%X6;
   IF #_w14 THEN #Events.%X6 := TRUE; END_IF;
   #ev := #_w14;
   IF #_w13 AND #Events.%X6 AND NOT #ev THEN #Events.%X6 := FALSE; END_IF;
   #_w15 := NOT #CMD.Local AND #pos[7];   // falling edge of #CMD.Local
   #pos[7] := #CMD.Local;
   #_w16 := #_w15 AND NOT #Events.%X7;
   IF #_w16 THEN #Events.%X7 := TRUE; END_IF;
   #ev := #_w16;
   IF #_w15 AND #Events.%X7 AND NOT #ev THEN #Events.%X7 := FALSE; END_IF;
   #_w17 := #CMD.Local AND #ON AND NOT #pos[8];   // rising edge of #ON
   #pos[8] := #ON;
   #_w18 := #_w17 AND NOT #Events.%X8;
   IF #_w18 THEN #Events.%X8 := TRUE; END_IF;
   #ev := #_w18;
   IF #_w17 AND #Events.%X8 AND NOT #ev THEN #Events.%X8 := FALSE; END_IF;
   #_w19 := #CMD.Local AND NOT #ON AND #pos[9];   // falling edge of #ON
   #pos[9] := #ON;
   #_w20 := #_w19 AND NOT #Events.%X9;
   IF #_w20 THEN #Events.%X9 := TRUE; END_IF;
   #ev := #_w20;
   IF #_w19 AND #Events.%X9 AND NOT #ev THEN #Events.%X9 := FALSE; END_IF;
   #_w21 := #CMD.Service AND NOT #pos[10];   // rising edge of #CMD.Service
   #pos[10] := #CMD.Service;
   #_w22 := #_w21 AND NOT #Events.%X10;
   IF #_w22 THEN #Events.%X10 := TRUE; END_IF;
   #ev := #_w22;
   IF #_w21 AND #Events.%X10 AND NOT #ev THEN #Events.%X10 := FALSE; END_IF;
   #_w23 := NOT #CMD.Service AND #pos[11];   // falling edge of #CMD.Service
   #pos[11] := #CMD.Service;
   #_w24 := #_w23 AND NOT #Events.%X11;
   IF #_w24 THEN #Events.%X11 := TRUE; END_IF;
   #ev := #_w24;
   IF #_w23 AND #Events.%X11 AND NOT #ev THEN #Events.%X11 := FALSE; END_IF;
   #_w25 := #CMD.ResetOpTime AND NOT #pos[12];   // rising edge of #CMD.ResetOpTime
   #pos[12] := #CMD.ResetOpTime;
   #_w26 := #_w25 AND NOT #Events.%X12;
   IF #_w26 THEN #Events.%X12 := TRUE; END_IF;
   #ev := #_w26;
   IF #_w25 AND #Events.%X12 AND NOT #ev THEN #Events.%X12 := FALSE; END_IF;
END_REGION

REGION Network 31: Сервисный режим
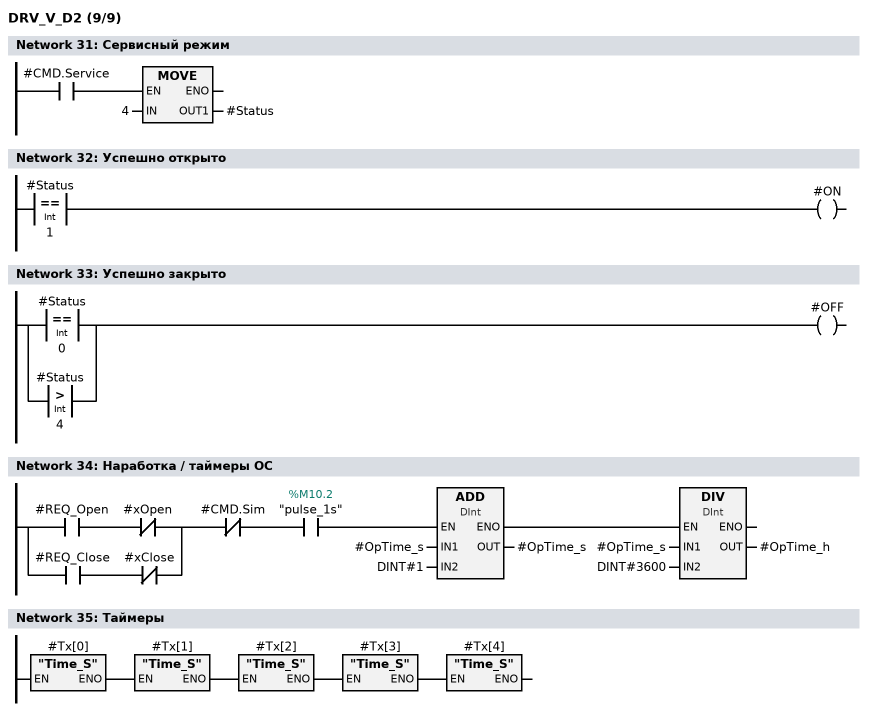
   RUNG wire#powerrail
      Contact( #CMD.Service )
      { S7_GenerateENO := "TRUE" } Move(in := 4, out1 => #Status)
   END_RUNG
   // the same network as SCL:
   IF #CMD.Service THEN #Status := 4; END_IF;
END_REGION

REGION Network 32: Успешно открыто
   RUNG wire#powerrail
      { S7_Templates := "SrcType := Int" } EQ_Contact(in1 := #Status, in2 := 1)
      Coil( #ON )
   END_RUNG
   // the same network as SCL:
   #ON := #Status = 1;
END_REGION

REGION Network 33: Успешно закрыто
   RUNG wire#powerrail
      { S7_Templates := "SrcType := Int" } EQ_Contact(in1 := #Status, in2 := 0)
      wire#w1
      Coil( #OFF )
   END_RUNG
   RUNG wire#powerrail
      { S7_Templates := "SrcType := Int" } GT_Contact(in1 := #Status, in2 := 4)
   END_RUNG wire#w1
   // the same network as SCL:
   #OFF := (#Status = 0) OR (#Status > 4);
END_REGION

REGION Network 34: Наработка / таймеры ОС
   RUNG wire#powerrail
      Contact( #REQ_Open )
      I_Contact( #xOpen )
      wire#w1
      I_Contact( #CMD.Sim )
      Contact( "pulse_1s" )
      { S7_Templates := "SrcType := DInt"; S7_GenerateENO := "TRUE" } Add(in1 := #OpTime_s, in2 := DINT#1, out => #OpTime_s)
      { S7_Templates := "SrcType := DInt"; S7_GenerateENO := "TRUE" } Div(in1 := #OpTime_s, in2 := DINT#3600, out => #OpTime_h)
   END_RUNG
   RUNG wire#powerrail
      Contact( #REQ_Close )
      I_Contact( #xClose )
   END_RUNG wire#w1
   // the same network as SCL:
   // ENO of a box is taken as its EN; it also drops when the box reports an error
   IF ((#REQ_Open AND NOT #xOpen) OR (#REQ_Close AND NOT #xClose)) AND NOT #CMD.Sim AND "pulse_1s" THEN
       #OpTime_s := #OpTime_s + DINT#1;
       #OpTime_h := #OpTime_s / DINT#3600;
   END_IF;
END_REGION

REGION Network 35: Таймеры
   RUNG wire#powerrail
      #Tx[0]()
      #Tx[1]()
      #Tx[2]()
      #Tx[3]()
      #Tx[4]()
   END_RUNG
   // the same network as SCL:
   #Tx[0](ENO => #_w1);   // "Time_S"
   #Tx[1](EN := #_w1, ENO => #_w2);   // "Time_S"
   #Tx[2](EN := #_w2, ENO => #_w3);   // "Time_S"
   #Tx[3](EN := #_w3, ENO => #_w4);   // "Time_S"
   IF #_w4 THEN
       #Tx[4]();   // "Time_S"
   END_IF;
END_REGION
END_FUNCTION_BLOCK

FUNCTION_BLOCK "DRV_V_D2A"   // FB121, LAD
TITLE = Управление клапаном с двумя дискретными положениями
{ S7_Optimized_Access := 'FALSE' }
VERSION : 0.1
// stored: AutoNumber false, IsIECCheckEnabled false, SetENOAutomatically false, UDAEnableTagReadback false
   VAR_INPUT
      All_Block : Bool;   // Аварийный останов
   END_VAR
   VAR_IN_OUT
      FB_QF : Bool;   // Защитный автомат
      FB_KM_Open : Bool;   // Пускатель - открыть
      FB_KM_Close : Bool;   // Пускатель - закрыть
      FB_Open : Bool;   // ОС - открыто
      FB_Close : Bool;   // ОС - закрыто
      S_Alarm : Bool;   // Наличие аварии
      CMD_Open : Bool;   // Команда - открыть
      CMD_Close : Bool;   // Команда - закрыть
   END_VAR
   VAR DB_SPECIFIC
      CMD : "CMD";   // Блок команд
      Mode : Int;   // Режим работы
      Status : Int;   // Статус устройства
      Use : Struct   // Функционал
         QF { S7_SetPoint := 'True'} : Bool;   // Защитный автомат
         KM_Open { S7_SetPoint := 'True'} : Bool;   // Пускатель - открыть
         KM_Close { S7_SetPoint := 'True'} : Bool;   // Пускатель - закрыть
         Open { S7_SetPoint := 'True'} : Bool := true;   // ОС - открыто
         Close { S7_SetPoint := 'True'} : Bool := true;   // ОС - закрыто
         One_KM { S7_SetPoint := 'True'} : Bool;   // Общий пускатель
         Electro { S7_SetPoint := 'True'} : Bool;   // Электропривод (остановка при срабатывании концевика)
         Cross { S7_SetPoint := 'True'} : Bool;   // Кросс-замена датчиков
         CMD_Open { S7_SetPoint := 'True'} : Bool := true;
         CMD_Close { S7_SetPoint := 'True'} : Bool;
         CMD_Reset { S7_SetPoint := 'True'} : Bool;
         calibration : Bool;
      END_STRUCT;
      FB : Struct   // Функционал
         Ready : Bool;   // Готовность к запуску
         QF : Bool;   // Защитный автомат
         KM_Open : Bool;   // Пускатель - открыть
         KM_Close : Bool;   // Пускатель - закрыть
         Open : Bool;   // ОС - открыто
         Close : Bool;   // ОС - закрыто
         Reserv : Bool;
         Local_Open : Bool;   // Локальное открытие
         Local_Close : Bool;   // Локальное закрытие
         pos_ok : Bool;   // положение достигнуто
         pos_open : Bool;   // клапан открывается
         pos_close : Bool;   // клапан закрывается
      END_STRUCT;
      ON : Bool;   // Успешно запущено
      OFF : Bool;   // Успешно остановлено
      REQ_Open : Bool;   // Запрос на открытие
      REQ_Close : Bool;   // Запрос на закрытие
   END_VAR
   VAR
      Tx { S7_SetPoint := 'True'} : Array[0..4] of "Time_S";   // Блок таймеров
   END_VAR
   VAR DB_SPECIFIC
      Inv : Struct   // Инверсия сигналов
         CMD { S7_SetPoint := 'True'} : Bool;   // Команда запуска
         QF { S7_SetPoint := 'True'} : Bool;   // Защитный автомат
         KM_Open { S7_SetPoint := 'True'} : Bool;   // Пускатель - открыть
         KM_Close { S7_SetPoint := 'True'} : Bool;   // Пускатель - закрыть
         Serivce { S7_SetPoint := 'True'} : Bool;   // Сервисный выключатель
         Open { S7_SetPoint := 'True'} : Bool;   // ОС - открыто
         Close { S7_SetPoint := 'True'} : Bool;   // ОС - закрыто
         Local_Open { S7_SetPoint := 'True'} : Bool;   // Локальное открытие
         Local_Close { S7_SetPoint := 'True'} : Bool;   // Локальное закрытие
      END_STRUCT;
      Alarm : Struct   // Список аварий
         Block : Bool;   // Аварийная остановка
         QF : Bool;   // Выбило защитный автомат
         KM_Open : Bool;   // Не сработал пускатель - открыть
         KM_Close : Bool;   // Не сработал пускатель - закрыть
         Two_S : Bool;   // Две ОС
         Open : Bool;   // Не сработал концевик - открыто
         Close : Bool;   // Не сработал концевик - закрыто
         OpTime : Bool;
      END_STRUCT;
      Alarms : Word;   // Слово аварий
      OpTime_h : DInt;   // наработка (ч)
      OpTime_s { S7_SetPoint := 'True'} : DInt;   // наработка (с)
      CodeID { S7_SetPoint := 'True'} : Int;   // Код датчика для привязки в скаде
      Indirect : Struct
         FB_QF { S7_SetPoint := 'True'} : Bool := true;   // Защитный автомат
         FB_KM_Open { S7_SetPoint := 'True'} : Bool := true;   // Пускатель - открыть
         FB_KM_Close { S7_SetPoint := 'True'} : Bool := true;   // Пускатель - закрыть
         FB_Open { S7_SetPoint := 'True'} : Bool := true;   // ОС - открыто
         FB_Close { S7_SetPoint := 'True'} : Bool := true;   // ОС - закрыто
         CMD_Open { S7_SetPoint := 'True'} : Bool := true;   // Команда на открытие
         CMD_Close { S7_SetPoint := 'True'} : Bool := true;   // Команда на закрытие
      END_STRUCT;
      Indirect_BYTE : Struct
         FB_QF { S7_SetPoint := 'True'} : Int;   // Защитный автомат
         FB_KM_Open { S7_SetPoint := 'True'} : Int;   // Пускатель - открыть
         FB_KM_Close { S7_SetPoint := 'True'} : Int;   // Пускатель - закрыть
         FB_Open { S7_SetPoint := 'True'} : Int;   // ОС - открыто
         FB_Close { S7_SetPoint := 'True'} : Int;   // ОС - закрыто
         CMD_Open { S7_SetPoint := 'True'} : Int;   // Команда на открытие
         CMD_Close { S7_SetPoint := 'True'} : Int;   // Команда на закрытие
         CMD_Reset : Int;
      END_STRUCT;
      Indirect_BIT : Struct
         FB_QF { S7_SetPoint := 'True'} : Int;   // Защитный автомат
         FB_KM_Open { S7_SetPoint := 'True'} : Int;   // Пускатель - открыть
         FB_KM_Close { S7_SetPoint := 'True'} : Int;   // Пускатель - закрыть
         FB_Open { S7_SetPoint := 'True'} : Int;   // ОС - открыто
         FB_Close { S7_SetPoint := 'True'} : Int;   // ОС - закрыто
         CMD_Open { S7_SetPoint := 'True'} : Int;   // Команда на открытие
         CMD_Close { S7_SetPoint := 'True'} : Int;   // Команда на закрытие
         CMD_Reset : Int;
      END_STRUCT;
   END_VAR
   VAR
      Tx_Sm { S7_SetPoint := 'True'} : Array[0..2] of "Time_S_b";   // Блок таймеров
      Tx_R { S7_SetPoint := 'True'} : Array[0..1] of "Time_R";   // Блок таймеров
   END_VAR
   VAR DB_SPECIFIC
      SP_A : Real;
      SP_M : Real;
      SP : Real;
      POSITION : Real;
      "step" : Int;
      DB { S7_SetPoint := 'True'} : Real := 1.0;
      pos : Array[0..15] of Bool;
   END_VAR
   VAR_TEMP
      xQF : Bool;
      xKM_Open : Bool;
      xKM_Close : Bool;
      xOpen : Bool;
      xClose : Bool;
      min : Real;
      max : Real;
   END_VAR
   VAR CONSTANT
      Pos_MIN : Real := 0.0;
      Pos_MAX : Real := 100.0;
   END_VAR
   VAR_TEMP   // added for the SCL form of the ladder/FBD networks
      _w1 : Bool;
      _w2 : Bool;
      _w3 : Bool;
      _w4 : Bool;
      _w5 : Bool;
      _w6 : Bool;
      _w7 : Bool;
   END_VAR
BEGIN

REGION Network 1: Режим глобальной симуляции
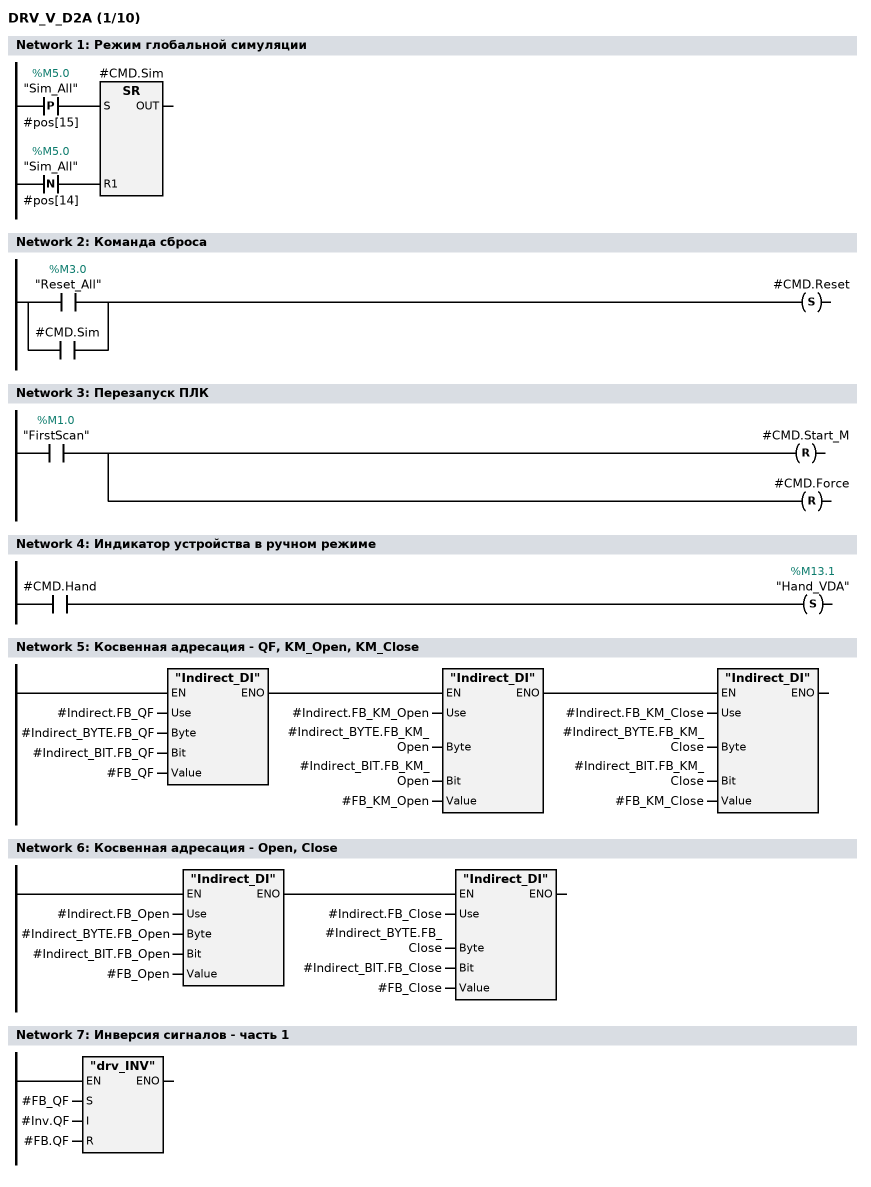
   RUNG wire#powerrail
      P_Contact(operand := "Sim_All", bit := #pos[15])
      S_SR(operand := #CMD.Sim, r1 := wire#w1)
   END_RUNG
   RUNG wire#powerrail
      N_Contact(operand := "Sim_All", bit := #pos[14])
   END_RUNG wire#w1
   // the same network as SCL:
   #_w1 := "Sim_All" AND NOT #pos[15];   // rising edge of "Sim_All"
   #pos[15] := "Sim_All";
   #_w2 := NOT "Sim_All" AND #pos[14];   // falling edge of "Sim_All"
   #pos[14] := "Sim_All";
   IF #_w1 THEN
       #CMD.Sim := TRUE;   // SR flip-flop
   END_IF;
   IF #_w2 THEN #CMD.Sim := FALSE; END_IF;
END_REGION

REGION Network 2: Команда сброса
   RUNG wire#powerrail
      Contact( "Reset_All" )
      wire#w1
      S_Coil( #CMD.Reset )
   END_RUNG
   RUNG wire#powerrail
      Contact( #CMD.Sim )
   END_RUNG wire#w1
   // the same network as SCL:
   IF "Reset_All" OR #CMD.Sim THEN #CMD.Reset := TRUE; END_IF;
END_REGION

REGION Network 3: Перезапуск ПЛК
   RUNG wire#powerrail
      Contact( "FirstScan" )
      wire#w1
      R_Coil( #CMD.Start_M )
   END_RUNG
   RUNG wire#w1
      R_Coil( #CMD.Force )
   END_RUNG
   // the same network as SCL:
   IF "FirstScan" THEN
       #CMD.Start_M := FALSE;
       #CMD.Force := FALSE;
   END_IF;
END_REGION

REGION Network 4: Индикатор устройства в ручном режиме
   RUNG wire#powerrail
      Contact( #CMD.Hand )
      S_Coil( "Hand_VDA" )
   END_RUNG
   // the same network as SCL:
   IF #CMD.Hand THEN "Hand_VDA" := TRUE; END_IF;
END_REGION

REGION Network 5: Косвенная адресация - QF, KM_Open, KM_Close
   RUNG wire#powerrail
      "Indirect_DI"(Use := #Indirect.FB_QF, "Byte" := #Indirect_BYTE.FB_QF, Bit := #Indirect_BIT.FB_QF, Value := #FB_QF)
      "Indirect_DI"(Use := #Indirect.FB_KM_Open, "Byte" := #Indirect_BYTE.FB_KM_Open, Bit := #Indirect_BIT.FB_KM_Open, Value := #FB_KM_Open)
      "Indirect_DI"(Use := #Indirect.FB_KM_Close, "Byte" := #Indirect_BYTE.FB_KM_Close, Bit := #Indirect_BIT.FB_KM_Close, Value := #FB_KM_Close)
   END_RUNG
   // the same network as SCL:
   "Indirect_DI"(Use := #Indirect.FB_QF,
                 "Byte" := #Indirect_BYTE.FB_QF,
                 Bit := #Indirect_BIT.FB_QF,
                 Value := #FB_QF,
                 ENO => #_w1);
   "Indirect_DI"(EN := #_w1,
                 Use := #Indirect.FB_KM_Open,
                 "Byte" := #Indirect_BYTE.FB_KM_Open,
                 Bit := #Indirect_BIT.FB_KM_Open,
                 Value := #FB_KM_Open,
                 ENO => #_w2);
   IF #_w2 THEN
       "Indirect_DI"(Use := #Indirect.FB_KM_Close,
                     "Byte" := #Indirect_BYTE.FB_KM_Close,
                     Bit := #Indirect_BIT.FB_KM_Close,
                     Value := #FB_KM_Close);
   END_IF;
END_REGION

REGION Network 6: Косвенная адресация - Open, Close
   RUNG wire#powerrail
      "Indirect_DI"(Use := #Indirect.FB_Open, "Byte" := #Indirect_BYTE.FB_Open, Bit := #Indirect_BIT.FB_Open, Value := #FB_Open)
      "Indirect_DI"(Use := #Indirect.FB_Close, "Byte" := #Indirect_BYTE.FB_Close, Bit := #Indirect_BIT.FB_Close, Value := #FB_Close)
   END_RUNG
   // the same network as SCL:
   "Indirect_DI"(Use := #Indirect.FB_Open,
                 "Byte" := #Indirect_BYTE.FB_Open,
                 Bit := #Indirect_BIT.FB_Open,
                 Value := #FB_Open,
                 ENO => #_w1);
   IF #_w1 THEN
       "Indirect_DI"(Use := #Indirect.FB_Close,
                     "Byte" := #Indirect_BYTE.FB_Close,
                     Bit := #Indirect_BIT.FB_Close,
                     Value := #FB_Close);
   END_IF;
END_REGION

REGION Network 7: Инверсия сигналов - часть 1
   RUNG wire#powerrail
      "drv_INV"(S := #FB_QF, I := #Inv.QF, R := #FB.QF)
   END_RUNG
   // the same network as SCL:
   "drv_INV"(S := #FB_QF, I := #Inv.QF, R := #FB.QF);
END_REGION

REGION Network 8: ОС
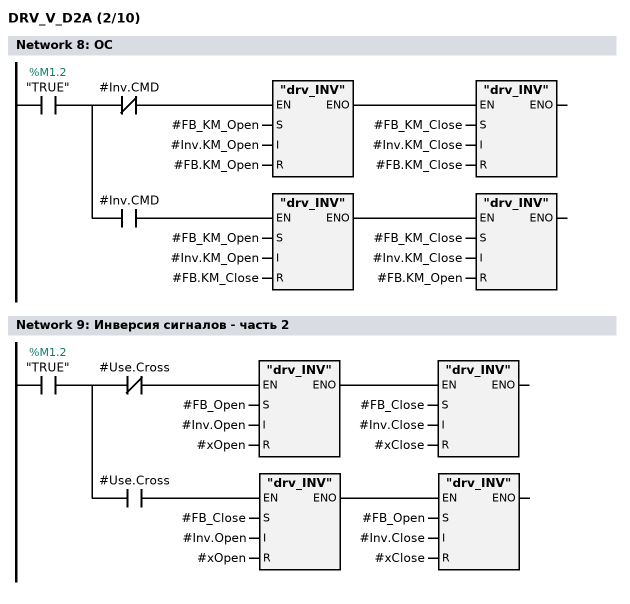
   RUNG wire#powerrail
      Contact( "TRUE" )
      wire#w1
      I_Contact( #Inv.CMD )
      "drv_INV"(S := #FB_KM_Open, I := #Inv.KM_Open, R := #FB.KM_Open)
      "drv_INV"(S := #FB_KM_Close, I := #Inv.KM_Close, R := #FB.KM_Close)
   END_RUNG
   RUNG wire#w1
      Contact( #Inv.CMD )
      "drv_INV"(S := #FB_KM_Open, I := #Inv.KM_Open, R := #FB.KM_Close)
      "drv_INV"(S := #FB_KM_Close, I := #Inv.KM_Close, R := #FB.KM_Open)
   END_RUNG
   // the same network as SCL:
   #_w2 := "TRUE";
   "drv_INV"(EN := "TRUE" AND NOT #Inv.CMD, S := #FB_KM_Open, I := #Inv.KM_Open, R := #FB.KM_Open, ENO => #_w1);
   IF #_w1 THEN "drv_INV"(S := #FB_KM_Close, I := #Inv.KM_Close, R := #FB.KM_Close); END_IF;
   "drv_INV"(EN := #_w2 AND #Inv.CMD, S := #FB_KM_Open, I := #Inv.KM_Open, R := #FB.KM_Close, ENO => #_w3);
   IF #_w3 THEN "drv_INV"(S := #FB_KM_Close, I := #Inv.KM_Close, R := #FB.KM_Open); END_IF;
END_REGION

REGION Network 9: Инверсия сигналов - часть 2
   RUNG wire#powerrail
      Contact( "TRUE" )
      wire#w1
      I_Contact( #Use.Cross )
      "drv_INV"(S := #FB_Open, I := #Inv.Open, R := #xOpen)
      "drv_INV"(S := #FB_Close, I := #Inv.Close, R := #xClose)
   END_RUNG
   RUNG wire#w1
      Contact( #Use.Cross )
      "drv_INV"(S := #FB_Close, I := #Inv.Open, R := #xOpen)
      "drv_INV"(S := #FB_Open, I := #Inv.Close, R := #xClose)
   END_RUNG
   // the same network as SCL:
   #_w2 := "TRUE";
   "drv_INV"(EN := "TRUE" AND NOT #Use.Cross, S := #FB_Open, I := #Inv.Open, R := #xOpen, ENO => #_w1);
   IF #_w1 THEN "drv_INV"(S := #FB_Close, I := #Inv.Close, R := #xClose); END_IF;
   "drv_INV"(EN := #_w2 AND #Use.Cross, S := #FB_Close, I := #Inv.Open, R := #xOpen, ENO => #_w3);
   IF #_w3 THEN "drv_INV"(S := #FB_Open, I := #Inv.Close, R := #xClose); END_IF;
END_REGION

REGION Network 10: Заглушка индикаторов ОС
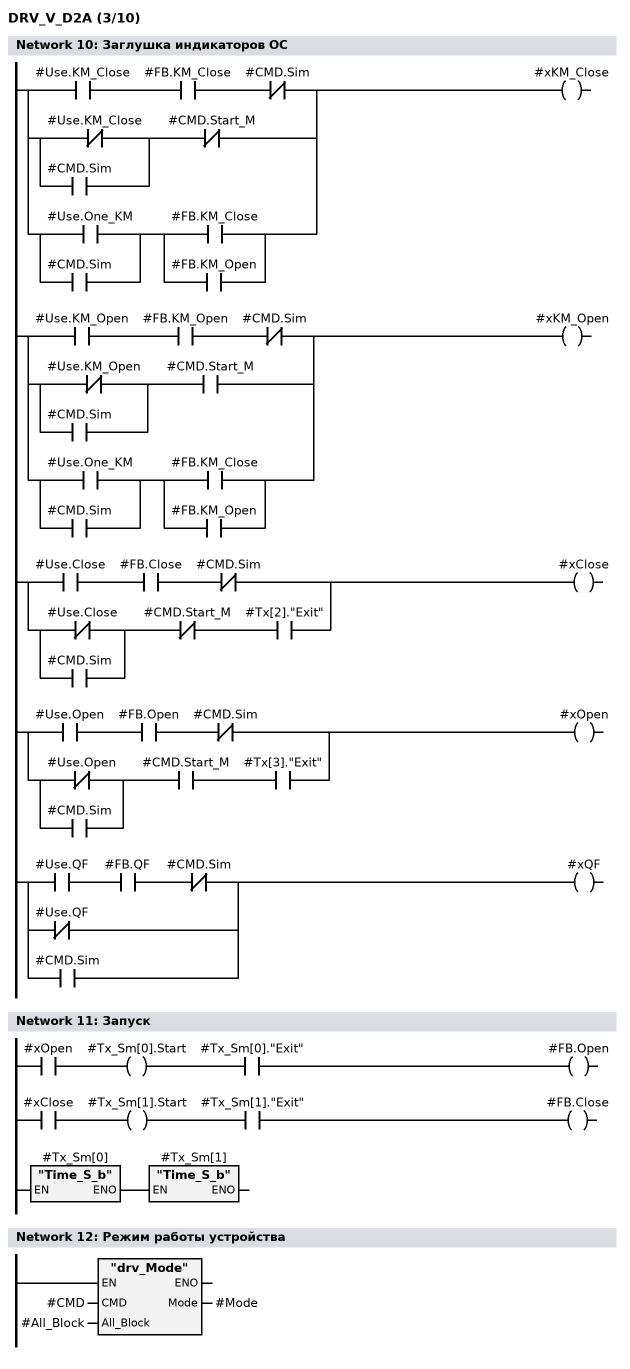
   RUNG wire#powerrail
      Contact( #Use.KM_Close )
      Contact( #FB.KM_Close )
      I_Contact( #CMD.Sim )
      wire#w1
      Coil( #xKM_Close )
   END_RUNG
   RUNG wire#powerrail
      I_Contact( #Use.KM_Close )
      wire#w2
      I_Contact( #CMD.Start_M )
   END_RUNG wire#w1
   RUNG wire#powerrail
      Contact( #CMD.Sim )
   END_RUNG wire#w2
   RUNG wire#powerrail
      Contact( #Use.One_KM )
      wire#w3
      Contact( #FB.KM_Close )
   END_RUNG wire#w1
   RUNG wire#powerrail
      Contact( #CMD.Sim )
   END_RUNG wire#w3
   RUNG wire#w3
      Contact( #FB.KM_Open )
   END_RUNG wire#w1
   RUNG wire#powerrail
      Contact( #Use.KM_Open )
      Contact( #FB.KM_Open )
      I_Contact( #CMD.Sim )
      wire#w4
      Coil( #xKM_Open )
   END_RUNG
   RUNG wire#powerrail
      I_Contact( #Use.KM_Open )
      wire#w5
      Contact( #CMD.Start_M )
   END_RUNG wire#w4
   RUNG wire#powerrail
      Contact( #CMD.Sim )
   END_RUNG wire#w5
   RUNG wire#powerrail
      Contact( #Use.One_KM )
      wire#w6
      Contact( #FB.KM_Close )
   END_RUNG wire#w4
   RUNG wire#powerrail
      Contact( #CMD.Sim )
   END_RUNG wire#w6
   RUNG wire#w6
      Contact( #FB.KM_Open )
   END_RUNG wire#w4
   RUNG wire#powerrail
      Contact( #Use.Close )
      Contact( #FB.Close )
      I_Contact( #CMD.Sim )
      wire#w7
      Coil( #xClose )
   END_RUNG
   RUNG wire#powerrail
      I_Contact( #Use.Close )
      wire#w8
      I_Contact( #CMD.Start_M )
      Contact( #Tx[2]."Exit" )
   END_RUNG wire#w7
   RUNG wire#powerrail
      Contact( #CMD.Sim )
   END_RUNG wire#w8
   RUNG wire#powerrail
      Contact( #Use.Open )
      Contact( #FB.Open )
      I_Contact( #CMD.Sim )
      wire#w9
      Coil( #xOpen )
   END_RUNG
   RUNG wire#powerrail
      I_Contact( #Use.Open )
      wire#w10
      Contact( #CMD.Start_M )
      Contact( #Tx[3]."Exit" )
   END_RUNG wire#w9
   RUNG wire#powerrail
      Contact( #CMD.Sim )
   END_RUNG wire#w10
   RUNG wire#powerrail
      Contact( #Use.QF )
      Contact( #FB.QF )
      I_Contact( #CMD.Sim )
      wire#w11
      Coil( #xQF )
   END_RUNG
   RUNG wire#powerrail
      I_Contact( #Use.QF )
   END_RUNG wire#w11
   RUNG wire#powerrail
      Contact( #CMD.Sim )
   END_RUNG wire#w11
   // the same network as SCL:
   #xKM_Close := (#Use.KM_Close AND #FB.KM_Close AND NOT #CMD.Sim) OR ((NOT #Use.KM_Close OR #CMD.Sim) AND NOT #CMD.Start_M) OR ((#Use.One_KM OR #CMD.Sim) AND (#FB.KM_Close OR #FB.KM_Open));
   #xKM_Open := (#Use.KM_Open AND #FB.KM_Open AND NOT #CMD.Sim) OR ((NOT #Use.KM_Open OR #CMD.Sim) AND #CMD.Start_M) OR ((#Use.One_KM OR #CMD.Sim) AND (#FB.KM_Close OR #FB.KM_Open));
   #xClose := (#Use.Close AND #FB.Close AND NOT #CMD.Sim) OR ((NOT #Use.Close OR #CMD.Sim) AND NOT #CMD.Start_M AND #Tx[2]."Exit");
   #xOpen := (#Use.Open AND #FB.Open AND NOT #CMD.Sim) OR ((NOT #Use.Open OR #CMD.Sim) AND #CMD.Start_M AND #Tx[3]."Exit");
   #xQF := (#Use.QF AND #FB.QF AND NOT #CMD.Sim) OR NOT #Use.QF OR #CMD.Sim;
END_REGION

REGION Network 11: Запуск
   RUNG wire#powerrail
      Contact( #xOpen )
      Coil( #Tx_Sm[0].Start )
      Contact( #Tx_Sm[0]."Exit" )
      Coil( #FB.Open )
   END_RUNG
   RUNG wire#powerrail
      Contact( #xClose )
      Coil( #Tx_Sm[1].Start )
      Contact( #Tx_Sm[1]."Exit" )
      Coil( #FB.Close )
   END_RUNG
   RUNG wire#powerrail
      #Tx_Sm[0]()
      #Tx_Sm[1]()
   END_RUNG
   // the same network as SCL:
   #Tx_Sm[0].Start := #xOpen;
   #FB.Open := #xOpen AND #Tx_Sm[0]."Exit";
   #Tx_Sm[1].Start := #xClose;
   #FB.Close := #xClose AND #Tx_Sm[1]."Exit";
   #Tx_Sm[0](ENO => #_w1);   // "Time_S_b"
   IF #_w1 THEN
       #Tx_Sm[1]();   // "Time_S_b"
   END_IF;
END_REGION

REGION Network 12: Режим работы устройства
   RUNG wire#powerrail
      "drv_Mode"(CMD := #CMD, All_Block := #All_Block, Mode => #Mode)
   END_RUNG
   // the same network as SCL:
   "drv_Mode"(CMD := #CMD, All_Block := #All_Block, Mode => #Mode);
END_REGION

REGION Network 13: Управление запуском
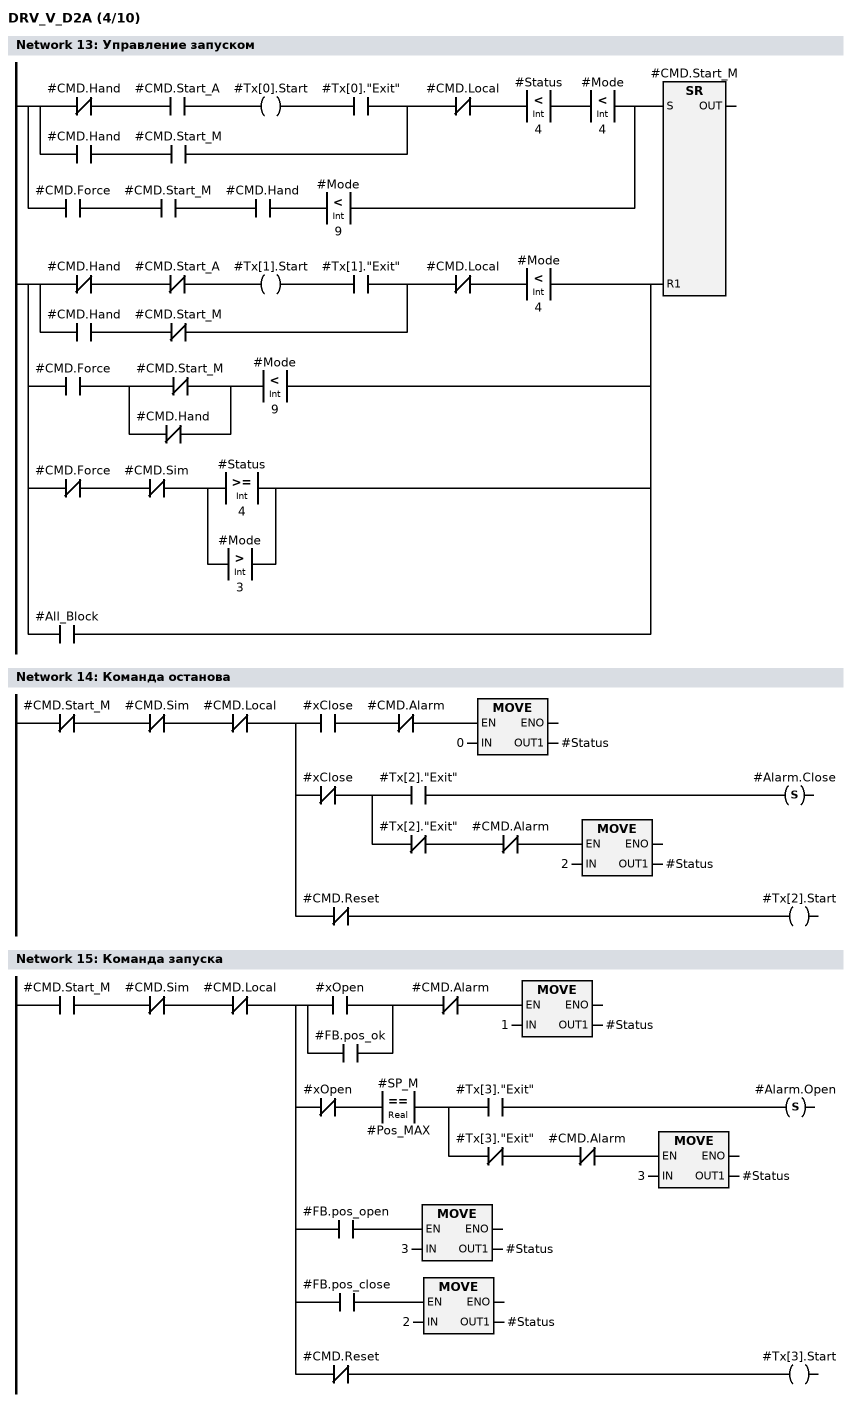
   RUNG wire#powerrail
      I_Contact( #CMD.Hand )
      Contact( #CMD.Start_A )
      Coil( #Tx[0].Start )
      Contact( #Tx[0]."Exit" )
      wire#w1
      I_Contact( #CMD.Local )
      { S7_Templates := "SrcType := Int" } LT_Contact(in1 := #Status, in2 := 4)
      { S7_Templates := "SrcType := Int" } LT_Contact(in1 := #Mode, in2 := 4)
      wire#w2
      S_SR(operand := #CMD.Start_M, r1 := wire#w7)
   END_RUNG
   RUNG wire#powerrail
      Contact( #CMD.Hand )
      Contact( #CMD.Start_M )
   END_RUNG wire#w1
   RUNG wire#powerrail
      Contact( #CMD.Force )
      Contact( #CMD.Start_M )
      Contact( #CMD.Hand )
      { S7_Templates := "SrcType := Int" } LT_Contact(in1 := #Mode, in2 := 9)
   END_RUNG wire#w2
   RUNG wire#powerrail
      I_Contact( #CMD.Hand )
      I_Contact( #CMD.Start_A )
      Coil( #Tx[1].Start )
      Contact( #Tx[1]."Exit" )
      wire#w3
      I_Contact( #CMD.Local )
      { S7_Templates := "SrcType := Int" } LT_Contact(in1 := #Mode, in2 := 4)
   END_RUNG wire#w7
   RUNG wire#powerrail
      Contact( #CMD.Hand )
      I_Contact( #CMD.Start_M )
   END_RUNG wire#w3
   RUNG wire#powerrail
      Contact( #CMD.Force )
      wire#w4
      I_Contact( #CMD.Start_M )
      wire#w5
      { S7_Templates := "SrcType := Int" } LT_Contact(in1 := #Mode, in2 := 9)
   END_RUNG wire#w7
   RUNG wire#w4
      I_Contact( #CMD.Hand )
   END_RUNG wire#w5
   RUNG wire#powerrail
      I_Contact( #CMD.Force )
      I_Contact( #CMD.Sim )
      wire#w6
      { S7_Templates := "SrcType := Int" } GE_Contact(in1 := #Status, in2 := 4)
   END_RUNG wire#w7
   RUNG wire#w6
      { S7_Templates := "SrcType := Int" } GT_Contact(in1 := #Mode, in2 := 3)
   END_RUNG wire#w7
   RUNG wire#powerrail
      Contact( #All_Block )
   END_RUNG wire#w7
   // the same network as SCL:
   #Tx[0].Start := NOT #CMD.Hand AND #CMD.Start_A;
   #_w1 := (((NOT #CMD.Hand AND #CMD.Start_A AND #Tx[0]."Exit") OR (#CMD.Hand AND #CMD.Start_M)) AND NOT #CMD.Local AND (#Status < 4) AND (#Mode < 4)) OR (#CMD.Force AND #CMD.Start_M AND #CMD.Hand AND (#Mode < 9));
   #Tx[1].Start := NOT #CMD.Hand AND NOT #CMD.Start_A;
   #_w2 := (((NOT #CMD.Hand AND NOT #CMD.Start_A AND #Tx[1]."Exit") OR (#CMD.Hand AND NOT #CMD.Start_M)) AND NOT #CMD.Local AND (#Mode < 4)) OR (#CMD.Force AND (NOT #CMD.Start_M OR NOT #CMD.Hand) AND (#Mode < 9)) OR (NOT #CMD.Force AND NOT #CMD.Sim AND ((#Status >= 4) OR (#Mode > 3))) OR #All_Block;
   IF #_w1 THEN
       #CMD.Start_M := TRUE;   // SR flip-flop
   END_IF;
   IF #_w2 THEN #CMD.Start_M := FALSE; END_IF;
END_REGION

REGION Network 14: Команда останова
   RUNG wire#powerrail
      I_Contact( #CMD.Start_M )
      I_Contact( #CMD.Sim )
      I_Contact( #CMD.Local )
      wire#w1
      Contact( #xClose )
      I_Contact( #CMD.Alarm )
      { S7_GenerateENO := "TRUE" } Move(in := 0, out1 => #Status)
   END_RUNG
   RUNG wire#w1
      I_Contact( #xClose )
      wire#w2
      Contact( #Tx[2]."Exit" )
      S_Coil( #Alarm.Close )
   END_RUNG
   RUNG wire#w2
      I_Contact( #Tx[2]."Exit" )
      I_Contact( #CMD.Alarm )
      { S7_GenerateENO := "TRUE" } Move(in := 2, out1 => #Status)
   END_RUNG
   RUNG wire#w1
      I_Contact( #CMD.Reset )
      Coil( #Tx[2].Start )
   END_RUNG
   // the same network as SCL:
   #_w1 := NOT #CMD.Start_M AND NOT #CMD.Sim AND NOT #CMD.Local;
   IF #_w1 AND #xClose AND NOT #CMD.Alarm THEN #Status := 0; END_IF;
   #_w2 := #_w1 AND NOT #xClose;
   IF #_w2 AND #Tx[2]."Exit" THEN #Alarm.Close := TRUE; END_IF;
   IF #_w2 AND NOT #Tx[2]."Exit" AND NOT #CMD.Alarm THEN #Status := 2; END_IF;
   #Tx[2].Start := #_w1 AND NOT #CMD.Reset;
END_REGION

REGION Network 15: Команда запуска
   RUNG wire#powerrail
      Contact( #CMD.Start_M )
      I_Contact( #CMD.Sim )
      I_Contact( #CMD.Local )
      wire#w1
      Contact( #xOpen )
      wire#w2
      I_Contact( #CMD.Alarm )
      { S7_GenerateENO := "TRUE" } Move(in := 1, out1 => #Status)
   END_RUNG
   RUNG wire#w1
      Contact( #FB.pos_ok )
   END_RUNG wire#w2
   RUNG wire#w1
      I_Contact( #xOpen )
      { S7_Templates := "SrcType := Real" } EQ_Contact(in1 := #SP_M, in2 := #Pos_MAX)
      wire#w3
      Contact( #Tx[3]."Exit" )
      S_Coil( #Alarm.Open )
   END_RUNG
   RUNG wire#w3
      I_Contact( #Tx[3]."Exit" )
      I_Contact( #CMD.Alarm )
      { S7_GenerateENO := "TRUE" } Move(in := 3, out1 => #Status)
   END_RUNG
   RUNG wire#w1
      Contact( #FB.pos_open )
      { S7_GenerateENO := "TRUE" } Move(in := 3, out1 => #Status)
   END_RUNG
   RUNG wire#w1
      Contact( #FB.pos_close )
      { S7_GenerateENO := "TRUE" } Move(in := 2, out1 => #Status)
   END_RUNG
   RUNG wire#w1
      I_Contact( #CMD.Reset )
      Coil( #Tx[3].Start )
   END_RUNG
   // the same network as SCL:
   #_w1 := #CMD.Start_M AND NOT #CMD.Sim AND NOT #CMD.Local;
   IF #_w1 AND (#xOpen OR #FB.pos_ok) AND NOT #CMD.Alarm THEN #Status := 1; END_IF;
   #_w2 := #_w1 AND NOT #xOpen AND (#SP_M = #Pos_MAX);
   IF #_w2 AND #Tx[3]."Exit" THEN #Alarm.Open := TRUE; END_IF;
   IF #_w2 AND NOT #Tx[3]."Exit" AND NOT #CMD.Alarm THEN #Status := 3; END_IF;
   IF #_w1 AND #FB.pos_open THEN #Status := 3; END_IF;
   IF #_w1 AND #FB.pos_close THEN #Status := 2; END_IF;
   #Tx[3].Start := #_w1 AND NOT #CMD.Reset;
END_REGION

REGION Network 16: Запрос на открытие
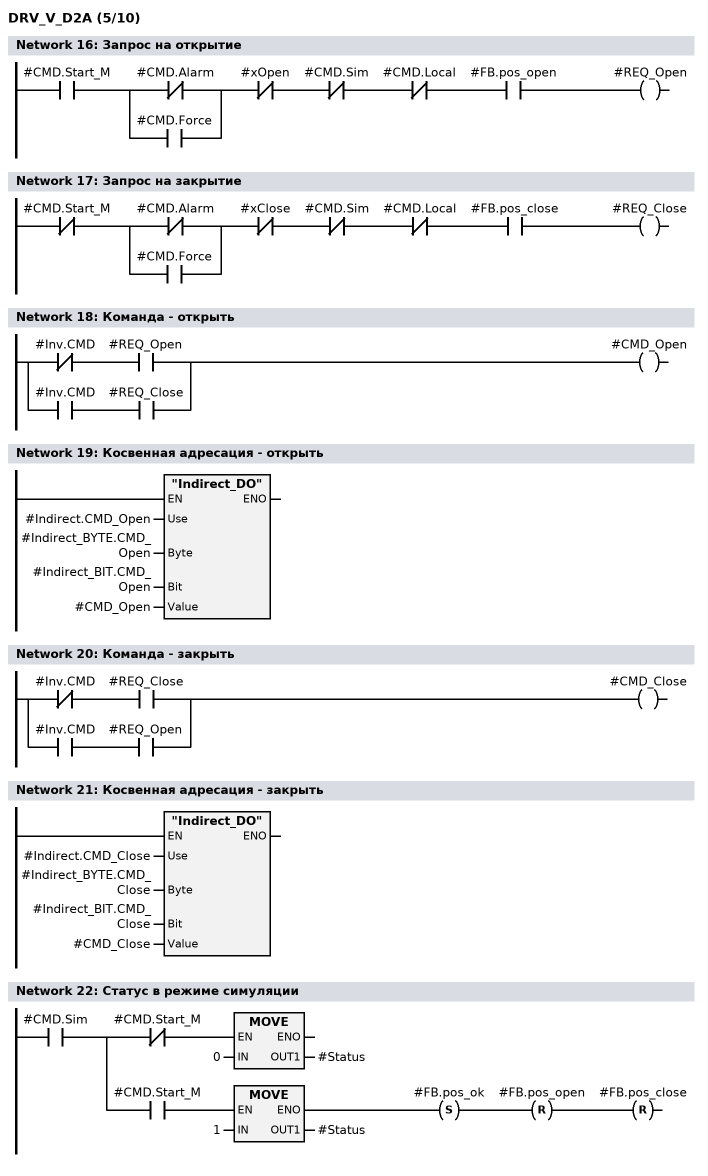
   RUNG wire#powerrail
      Contact( #CMD.Start_M )
      wire#w1
      I_Contact( #CMD.Alarm )
      wire#w2
      I_Contact( #xOpen )
      I_Contact( #CMD.Sim )
      I_Contact( #CMD.Local )
      Contact( #FB.pos_open )
      Coil( #REQ_Open )
   END_RUNG
   RUNG wire#w1
      Contact( #CMD.Force )
   END_RUNG wire#w2
   // the same network as SCL:
   #REQ_Open := #CMD.Start_M AND (NOT #CMD.Alarm OR #CMD.Force) AND NOT #xOpen AND NOT #CMD.Sim AND NOT #CMD.Local AND #FB.pos_open;
END_REGION

REGION Network 17: Запрос на закрытие
   RUNG wire#powerrail
      I_Contact( #CMD.Start_M )
      wire#w1
      I_Contact( #CMD.Alarm )
      wire#w2
      I_Contact( #xClose )
      I_Contact( #CMD.Sim )
      I_Contact( #CMD.Local )
      Contact( #FB.pos_close )
      Coil( #REQ_Close )
   END_RUNG
   RUNG wire#w1
      Contact( #CMD.Force )
   END_RUNG wire#w2
   // the same network as SCL:
   #REQ_Close := NOT #CMD.Start_M AND (NOT #CMD.Alarm OR #CMD.Force) AND NOT #xClose AND NOT #CMD.Sim AND NOT #CMD.Local AND #FB.pos_close;
END_REGION

REGION Network 18: Команда - открыть
   RUNG wire#powerrail
      I_Contact( #Inv.CMD )
      Contact( #REQ_Open )
      wire#w1
      Coil( #CMD_Open )
   END_RUNG
   RUNG wire#powerrail
      Contact( #Inv.CMD )
      Contact( #REQ_Close )
   END_RUNG wire#w1
   // the same network as SCL:
   #CMD_Open := (NOT #Inv.CMD AND #REQ_Open) OR (#Inv.CMD AND #REQ_Close);
END_REGION

REGION Network 19: Косвенная адресация - открыть
   RUNG wire#powerrail
      "Indirect_DO"(Use := #Indirect.CMD_Open, "Byte" := #Indirect_BYTE.CMD_Open, Bit := #Indirect_BIT.CMD_Open, Value := #CMD_Open)
   END_RUNG
   // the same network as SCL:
   "Indirect_DO"(Use := #Indirect.CMD_Open,
                 "Byte" := #Indirect_BYTE.CMD_Open,
                 Bit := #Indirect_BIT.CMD_Open,
                 Value := #CMD_Open);
END_REGION

REGION Network 20: Команда - закрыть
   RUNG wire#powerrail
      I_Contact( #Inv.CMD )
      Contact( #REQ_Close )
      wire#w1
      Coil( #CMD_Close )
   END_RUNG
   RUNG wire#powerrail
      Contact( #Inv.CMD )
      Contact( #REQ_Open )
   END_RUNG wire#w1
   // the same network as SCL:
   #CMD_Close := (NOT #Inv.CMD AND #REQ_Close) OR (#Inv.CMD AND #REQ_Open);
END_REGION

REGION Network 21: Косвенная адресация - закрыть
   RUNG wire#powerrail
      "Indirect_DO"(Use := #Indirect.CMD_Close, "Byte" := #Indirect_BYTE.CMD_Close, Bit := #Indirect_BIT.CMD_Close, Value := #CMD_Close)
   END_RUNG
   // the same network as SCL:
   "Indirect_DO"(Use := #Indirect.CMD_Close,
                 "Byte" := #Indirect_BYTE.CMD_Close,
                 Bit := #Indirect_BIT.CMD_Close,
                 Value := #CMD_Close);
END_REGION

